// TIA Portal V18 export
// export: Created 2026-06-12T02:00:00Z, ExportSetting WithDefaults
FUNCTION "FC_SCADA_Sim_B3to7" : Void   // FC11, LAD
{ S7_Optimized_Access := 'TRUE' }
VERSION : 0.1
// stored: AutoNumber true, IsIECCheckEnabled false
BEGIN

REGION Network 1: Tạo xung kích hoạt chu kỳ mô phỏng (50ms)
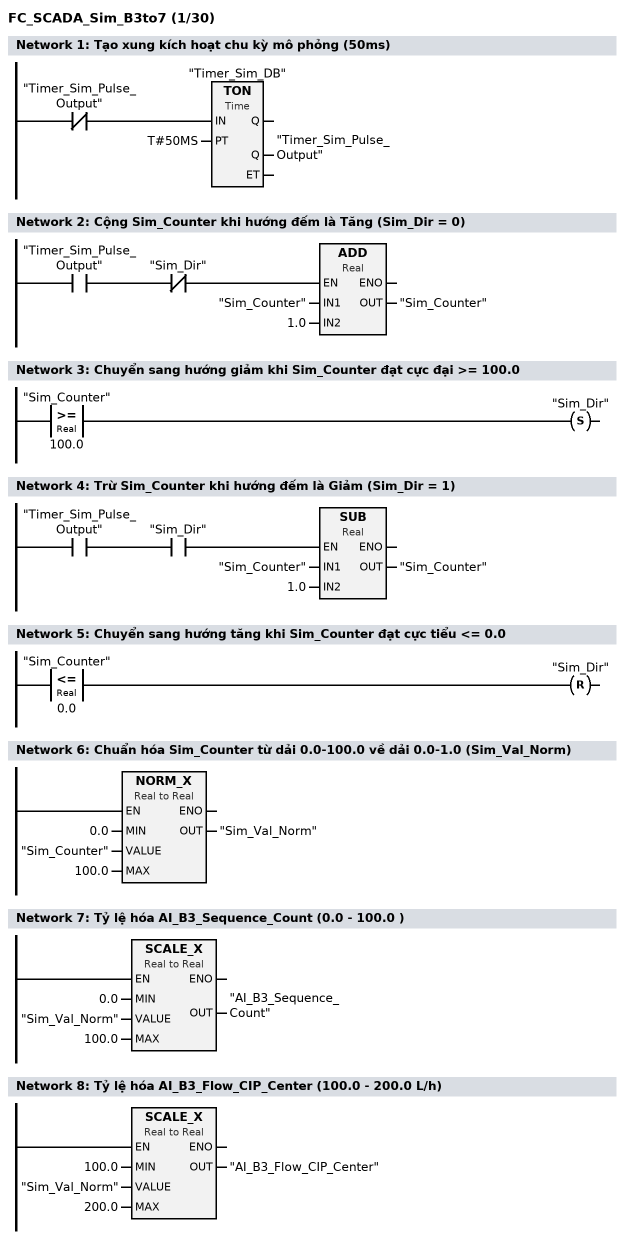
   RUNG wire#powerrail
      I_Contact( "Timer_Sim_Pulse_Output" )
      { S7_Templates := "time_type := Time" } "Timer_Sim_DB".TON(pt := T#50MS, q => "Timer_Sim_Pulse_Output", et =>)
   END_RUNG
   // the same network as SCL:
   "Timer_Sim_DB".TON(IN := NOT "Timer_Sim_Pulse_Output", PT := T#50MS, Q => "Timer_Sim_Pulse_Output");
END_REGION

REGION Network 2: Cộng Sim_Counter khi hướng đếm là Tăng (Sim_Dir = 0)
   RUNG wire#powerrail
      Contact( "Timer_Sim_Pulse_Output" )
      I_Contact( "Sim_Dir" )
      { S7_Templates := "SrcType := Real"; S7_GenerateENO := "TRUE" } Add(in1 := "Sim_Counter", in2 := 1.0, out => "Sim_Counter")
   END_RUNG
   // the same network as SCL:
   IF "Timer_Sim_Pulse_Output" AND NOT "Sim_Dir" THEN "Sim_Counter" := "Sim_Counter" + 1.0; END_IF;
END_REGION

REGION Network 3: Chuyển sang hướng giảm khi Sim_Counter đạt cực đại >= 100.0
   RUNG wire#powerrail
      { S7_Templates := "SrcType := Real" } GE_Contact(in1 := "Sim_Counter", in2 := 100.0)
      S_Coil( "Sim_Dir" )
   END_RUNG
   // the same network as SCL:
   IF "Sim_Counter" >= 100.0 THEN "Sim_Dir" := TRUE; END_IF;
END_REGION

REGION Network 4: Trừ Sim_Counter khi hướng đếm là Giảm (Sim_Dir = 1)
   RUNG wire#powerrail
      Contact( "Timer_Sim_Pulse_Output" )
      Contact( "Sim_Dir" )
      { S7_Templates := "SrcType := Real"; S7_GenerateENO := "TRUE" } Sub(in1 := "Sim_Counter", in2 := 1.0, out => "Sim_Counter")
   END_RUNG
   // the same network as SCL:
   IF "Timer_Sim_Pulse_Output" AND "Sim_Dir" THEN "Sim_Counter" := "Sim_Counter" - 1.0; END_IF;
END_REGION

REGION Network 5: Chuyển sang hướng tăng khi Sim_Counter đạt cực tiểu <= 0.0
   RUNG wire#powerrail
      { S7_Templates := "SrcType := Real" } LE_Contact(in1 := "Sim_Counter", in2 := 0.0)
      R_Coil( "Sim_Dir" )
   END_RUNG
   // the same network as SCL:
   IF "Sim_Counter" <= 0.0 THEN "Sim_Dir" := FALSE; END_IF;
END_REGION

REGION Network 6: Chuẩn hóa Sim_Counter từ dải 0.0-100.0 về dải 0.0-1.0 (Sim_Val_Norm)
   RUNG wire#powerrail
      { S7_Templates := "[SrcType := Real, DestType := Real]" } Normalize(min := 0.0, value := "Sim_Counter", max := 100.0, out => "Sim_Val_Norm")
   END_RUNG
   // the same network as SCL:
   "Sim_Val_Norm" := NORM_X(MIN := 0.0, VALUE := "Sim_Counter", MAX := 100.0);
END_REGION

REGION Network 7: Tỷ lệ hóa AI_B3_Sequence_Count (0.0 - 100.0 )
   RUNG wire#powerrail
      { S7_Templates := "[SrcType := Real, DestType := Real]" } Scale(min := 0.0, value := "Sim_Val_Norm", max := 100.0, out => "AI_B3_Sequence_Count")
   END_RUNG
   // the same network as SCL:
   "AI_B3_Sequence_Count" := SCALE_X(MIN := 0.0, VALUE := "Sim_Val_Norm", MAX := 100.0);
END_REGION

REGION Network 8: Tỷ lệ hóa AI_B3_Flow_CIP_Center (100.0 - 200.0 L/h)
   RUNG wire#powerrail
      { S7_Templates := "[SrcType := Real, DestType := Real]" } Scale(min := 100.0, value := "Sim_Val_Norm", max := 200.0, out => "AI_B3_Flow_CIP_Center")
   END_RUNG
   // the same network as SCL:
   "AI_B3_Flow_CIP_Center" := SCALE_X(MIN := 100.0, VALUE := "Sim_Val_Norm", MAX := 200.0);
END_REGION

REGION Network 9: Tỷ lệ hóa AI_B3_Temp_CIP_Upper (50.0 - 80.0 °C)
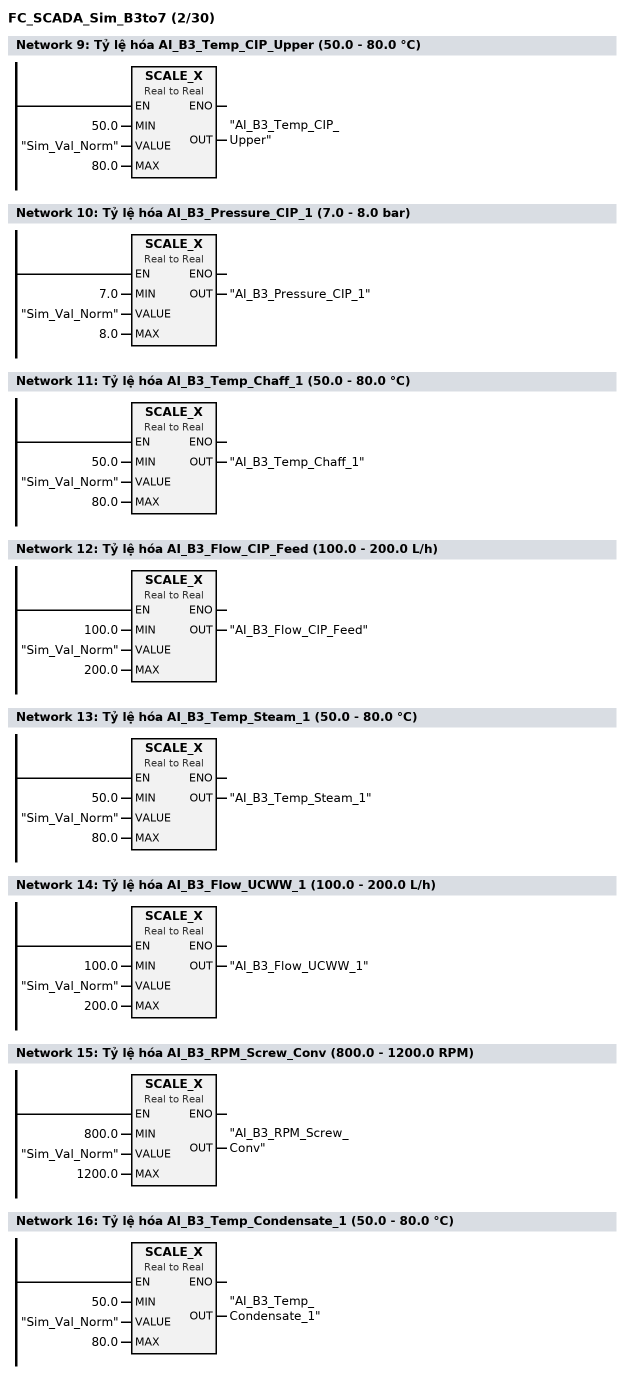
   RUNG wire#powerrail
      { S7_Templates := "[SrcType := Real, DestType := Real]" } Scale(min := 50.0, value := "Sim_Val_Norm", max := 80.0, out => "AI_B3_Temp_CIP_Upper")
   END_RUNG
   // the same network as SCL:
   "AI_B3_Temp_CIP_Upper" := SCALE_X(MIN := 50.0, VALUE := "Sim_Val_Norm", MAX := 80.0);
END_REGION

REGION Network 10: Tỷ lệ hóa AI_B3_Pressure_CIP_1 (7.0 - 8.0 bar)
   RUNG wire#powerrail
      { S7_Templates := "[SrcType := Real, DestType := Real]" } Scale(min := 7.0, value := "Sim_Val_Norm", max := 8.0, out => "AI_B3_Pressure_CIP_1")
   END_RUNG
   // the same network as SCL:
   "AI_B3_Pressure_CIP_1" := SCALE_X(MIN := 7.0, VALUE := "Sim_Val_Norm", MAX := 8.0);
END_REGION

REGION Network 11: Tỷ lệ hóa AI_B3_Temp_Chaff_1 (50.0 - 80.0 °C)
   RUNG wire#powerrail
      { S7_Templates := "[SrcType := Real, DestType := Real]" } Scale(min := 50.0, value := "Sim_Val_Norm", max := 80.0, out => "AI_B3_Temp_Chaff_1")
   END_RUNG
   // the same network as SCL:
   "AI_B3_Temp_Chaff_1" := SCALE_X(MIN := 50.0, VALUE := "Sim_Val_Norm", MAX := 80.0);
END_REGION

REGION Network 12: Tỷ lệ hóa AI_B3_Flow_CIP_Feed (100.0 - 200.0 L/h)
   RUNG wire#powerrail
      { S7_Templates := "[SrcType := Real, DestType := Real]" } Scale(min := 100.0, value := "Sim_Val_Norm", max := 200.0, out => "AI_B3_Flow_CIP_Feed")
   END_RUNG
   // the same network as SCL:
   "AI_B3_Flow_CIP_Feed" := SCALE_X(MIN := 100.0, VALUE := "Sim_Val_Norm", MAX := 200.0);
END_REGION

REGION Network 13: Tỷ lệ hóa AI_B3_Temp_Steam_1 (50.0 - 80.0 °C)
   RUNG wire#powerrail
      { S7_Templates := "[SrcType := Real, DestType := Real]" } Scale(min := 50.0, value := "Sim_Val_Norm", max := 80.0, out => "AI_B3_Temp_Steam_1")
   END_RUNG
   // the same network as SCL:
   "AI_B3_Temp_Steam_1" := SCALE_X(MIN := 50.0, VALUE := "Sim_Val_Norm", MAX := 80.0);
END_REGION

REGION Network 14: Tỷ lệ hóa AI_B3_Flow_UCWW_1 (100.0 - 200.0 L/h)
   RUNG wire#powerrail
      { S7_Templates := "[SrcType := Real, DestType := Real]" } Scale(min := 100.0, value := "Sim_Val_Norm", max := 200.0, out => "AI_B3_Flow_UCWW_1")
   END_RUNG
   // the same network as SCL:
   "AI_B3_Flow_UCWW_1" := SCALE_X(MIN := 100.0, VALUE := "Sim_Val_Norm", MAX := 200.0);
END_REGION

REGION Network 15: Tỷ lệ hóa AI_B3_RPM_Screw_Conv (800.0 - 1200.0 RPM)
   RUNG wire#powerrail
      { S7_Templates := "[SrcType := Real, DestType := Real]" } Scale(min := 800.0, value := "Sim_Val_Norm", max := 1200.0, out => "AI_B3_RPM_Screw_Conv")
   END_RUNG
   // the same network as SCL:
   "AI_B3_RPM_Screw_Conv" := SCALE_X(MIN := 800.0, VALUE := "Sim_Val_Norm", MAX := 1200.0);
END_REGION

REGION Network 16: Tỷ lệ hóa AI_B3_Temp_Condensate_1 (50.0 - 80.0 °C)
   RUNG wire#powerrail
      { S7_Templates := "[SrcType := Real, DestType := Real]" } Scale(min := 50.0, value := "Sim_Val_Norm", max := 80.0, out => "AI_B3_Temp_Condensate_1")
   END_RUNG
   // the same network as SCL:
   "AI_B3_Temp_Condensate_1" := SCALE_X(MIN := 50.0, VALUE := "Sim_Val_Norm", MAX := 80.0);
END_REGION

REGION Network 17: Tỷ lệ hóa AI_B3_Pressure_Screw_1 (7.0 - 8.0 bar)
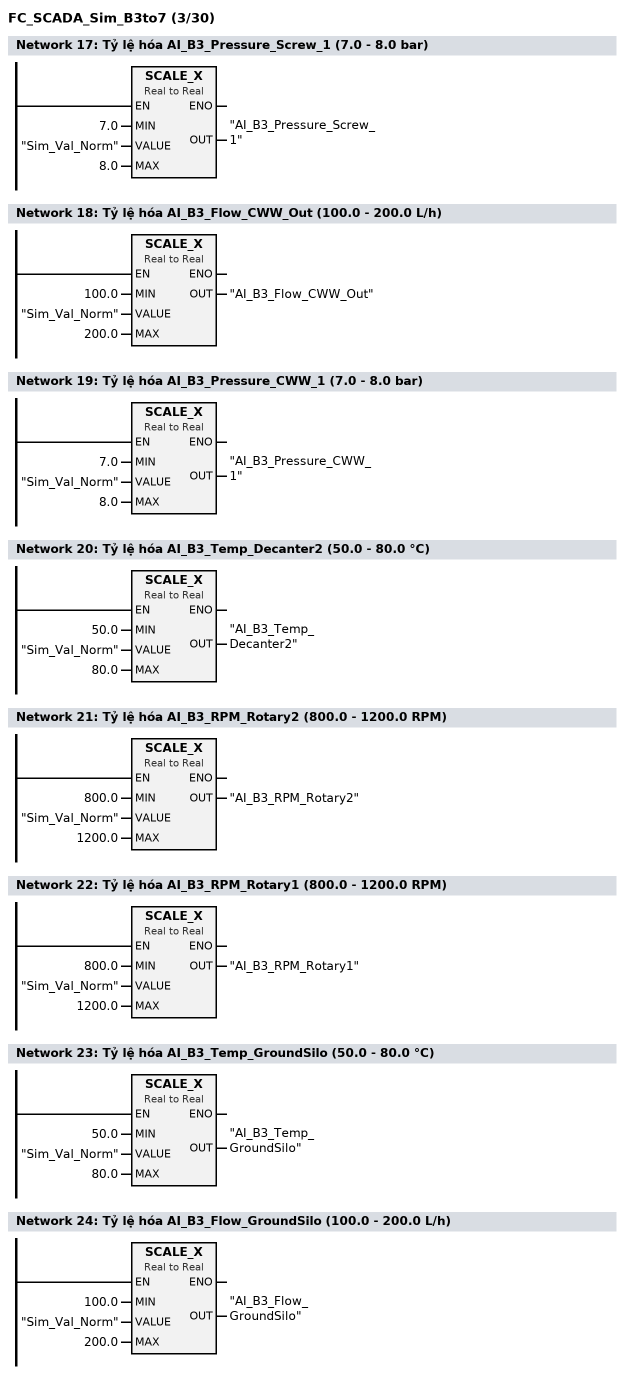
   RUNG wire#powerrail
      { S7_Templates := "[SrcType := Real, DestType := Real]" } Scale(min := 7.0, value := "Sim_Val_Norm", max := 8.0, out => "AI_B3_Pressure_Screw_1")
   END_RUNG
   // the same network as SCL:
   "AI_B3_Pressure_Screw_1" := SCALE_X(MIN := 7.0, VALUE := "Sim_Val_Norm", MAX := 8.0);
END_REGION

REGION Network 18: Tỷ lệ hóa AI_B3_Flow_CWW_Out (100.0 - 200.0 L/h)
   RUNG wire#powerrail
      { S7_Templates := "[SrcType := Real, DestType := Real]" } Scale(min := 100.0, value := "Sim_Val_Norm", max := 200.0, out => "AI_B3_Flow_CWW_Out")
   END_RUNG
   // the same network as SCL:
   "AI_B3_Flow_CWW_Out" := SCALE_X(MIN := 100.0, VALUE := "Sim_Val_Norm", MAX := 200.0);
END_REGION

REGION Network 19: Tỷ lệ hóa AI_B3_Pressure_CWW_1 (7.0 - 8.0 bar)
   RUNG wire#powerrail
      { S7_Templates := "[SrcType := Real, DestType := Real]" } Scale(min := 7.0, value := "Sim_Val_Norm", max := 8.0, out => "AI_B3_Pressure_CWW_1")
   END_RUNG
   // the same network as SCL:
   "AI_B3_Pressure_CWW_1" := SCALE_X(MIN := 7.0, VALUE := "Sim_Val_Norm", MAX := 8.0);
END_REGION

REGION Network 20: Tỷ lệ hóa AI_B3_Temp_Decanter2 (50.0 - 80.0 °C)
   RUNG wire#powerrail
      { S7_Templates := "[SrcType := Real, DestType := Real]" } Scale(min := 50.0, value := "Sim_Val_Norm", max := 80.0, out => "AI_B3_Temp_Decanter2")
   END_RUNG
   // the same network as SCL:
   "AI_B3_Temp_Decanter2" := SCALE_X(MIN := 50.0, VALUE := "Sim_Val_Norm", MAX := 80.0);
END_REGION

REGION Network 21: Tỷ lệ hóa AI_B3_RPM_Rotary2 (800.0 - 1200.0 RPM)
   RUNG wire#powerrail
      { S7_Templates := "[SrcType := Real, DestType := Real]" } Scale(min := 800.0, value := "Sim_Val_Norm", max := 1200.0, out => "AI_B3_RPM_Rotary2")
   END_RUNG
   // the same network as SCL:
   "AI_B3_RPM_Rotary2" := SCALE_X(MIN := 800.0, VALUE := "Sim_Val_Norm", MAX := 1200.0);
END_REGION

REGION Network 22: Tỷ lệ hóa AI_B3_RPM_Rotary1 (800.0 - 1200.0 RPM)
   RUNG wire#powerrail
      { S7_Templates := "[SrcType := Real, DestType := Real]" } Scale(min := 800.0, value := "Sim_Val_Norm", max := 1200.0, out => "AI_B3_RPM_Rotary1")
   END_RUNG
   // the same network as SCL:
   "AI_B3_RPM_Rotary1" := SCALE_X(MIN := 800.0, VALUE := "Sim_Val_Norm", MAX := 1200.0);
END_REGION

REGION Network 23: Tỷ lệ hóa AI_B3_Temp_GroundSilo (50.0 - 80.0 °C)
   RUNG wire#powerrail
      { S7_Templates := "[SrcType := Real, DestType := Real]" } Scale(min := 50.0, value := "Sim_Val_Norm", max := 80.0, out => "AI_B3_Temp_GroundSilo")
   END_RUNG
   // the same network as SCL:
   "AI_B3_Temp_GroundSilo" := SCALE_X(MIN := 50.0, VALUE := "Sim_Val_Norm", MAX := 80.0);
END_REGION

REGION Network 24: Tỷ lệ hóa AI_B3_Flow_GroundSilo (100.0 - 200.0 L/h)
   RUNG wire#powerrail
      { S7_Templates := "[SrcType := Real, DestType := Real]" } Scale(min := 100.0, value := "Sim_Val_Norm", max := 200.0, out => "AI_B3_Flow_GroundSilo")
   END_RUNG
   // the same network as SCL:
   "AI_B3_Flow_GroundSilo" := SCALE_X(MIN := 100.0, VALUE := "Sim_Val_Norm", MAX := 200.0);
END_REGION

REGION Network 25: Tỷ lệ hóa AI_B3_Pressure_Mid_1 (7.0 - 8.0 bar)
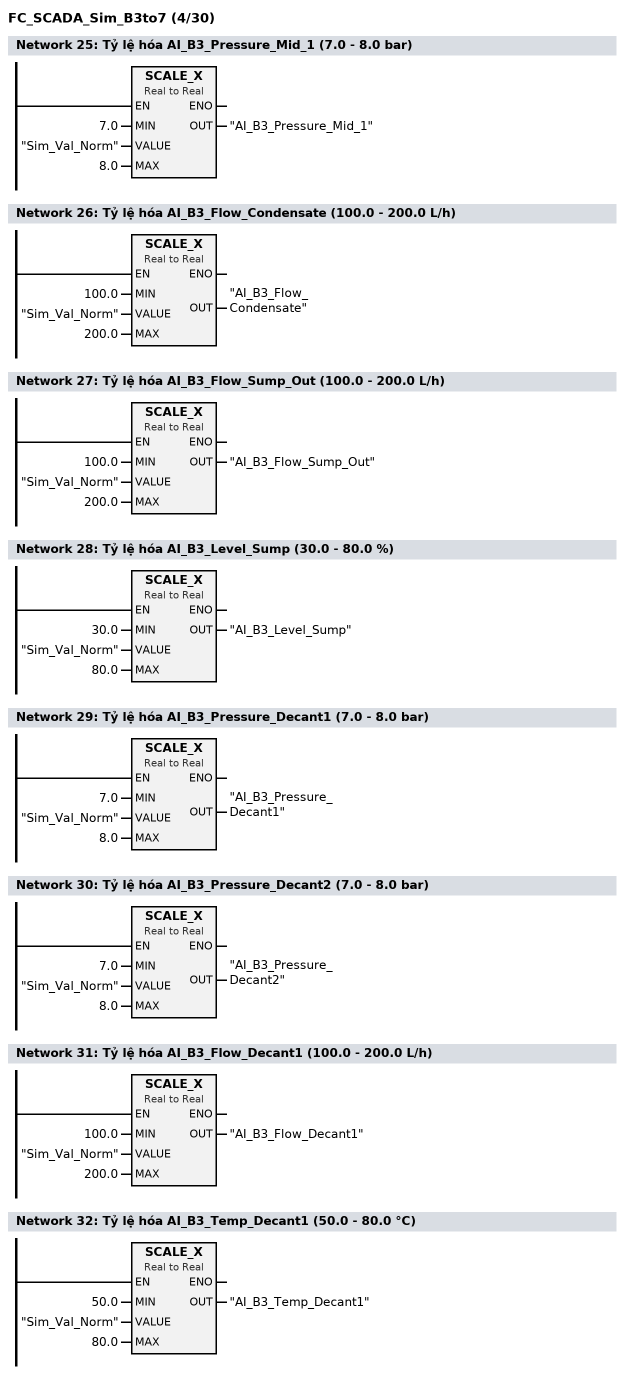
   RUNG wire#powerrail
      { S7_Templates := "[SrcType := Real, DestType := Real]" } Scale(min := 7.0, value := "Sim_Val_Norm", max := 8.0, out => "AI_B3_Pressure_Mid_1")
   END_RUNG
   // the same network as SCL:
   "AI_B3_Pressure_Mid_1" := SCALE_X(MIN := 7.0, VALUE := "Sim_Val_Norm", MAX := 8.0);
END_REGION

REGION Network 26: Tỷ lệ hóa AI_B3_Flow_Condensate (100.0 - 200.0 L/h)
   RUNG wire#powerrail
      { S7_Templates := "[SrcType := Real, DestType := Real]" } Scale(min := 100.0, value := "Sim_Val_Norm", max := 200.0, out => "AI_B3_Flow_Condensate")
   END_RUNG
   // the same network as SCL:
   "AI_B3_Flow_Condensate" := SCALE_X(MIN := 100.0, VALUE := "Sim_Val_Norm", MAX := 200.0);
END_REGION

REGION Network 27: Tỷ lệ hóa AI_B3_Flow_Sump_Out (100.0 - 200.0 L/h)
   RUNG wire#powerrail
      { S7_Templates := "[SrcType := Real, DestType := Real]" } Scale(min := 100.0, value := "Sim_Val_Norm", max := 200.0, out => "AI_B3_Flow_Sump_Out")
   END_RUNG
   // the same network as SCL:
   "AI_B3_Flow_Sump_Out" := SCALE_X(MIN := 100.0, VALUE := "Sim_Val_Norm", MAX := 200.0);
END_REGION

REGION Network 28: Tỷ lệ hóa AI_B3_Level_Sump (30.0 - 80.0 %)
   RUNG wire#powerrail
      { S7_Templates := "[SrcType := Real, DestType := Real]" } Scale(min := 30.0, value := "Sim_Val_Norm", max := 80.0, out => "AI_B3_Level_Sump")
   END_RUNG
   // the same network as SCL:
   "AI_B3_Level_Sump" := SCALE_X(MIN := 30.0, VALUE := "Sim_Val_Norm", MAX := 80.0);
END_REGION

REGION Network 29: Tỷ lệ hóa AI_B3_Pressure_Decant1 (7.0 - 8.0 bar)
   RUNG wire#powerrail
      { S7_Templates := "[SrcType := Real, DestType := Real]" } Scale(min := 7.0, value := "Sim_Val_Norm", max := 8.0, out => "AI_B3_Pressure_Decant1")
   END_RUNG
   // the same network as SCL:
   "AI_B3_Pressure_Decant1" := SCALE_X(MIN := 7.0, VALUE := "Sim_Val_Norm", MAX := 8.0);
END_REGION

REGION Network 30: Tỷ lệ hóa AI_B3_Pressure_Decant2 (7.0 - 8.0 bar)
   RUNG wire#powerrail
      { S7_Templates := "[SrcType := Real, DestType := Real]" } Scale(min := 7.0, value := "Sim_Val_Norm", max := 8.0, out => "AI_B3_Pressure_Decant2")
   END_RUNG
   // the same network as SCL:
   "AI_B3_Pressure_Decant2" := SCALE_X(MIN := 7.0, VALUE := "Sim_Val_Norm", MAX := 8.0);
END_REGION

REGION Network 31: Tỷ lệ hóa AI_B3_Flow_Decant1 (100.0 - 200.0 L/h)
   RUNG wire#powerrail
      { S7_Templates := "[SrcType := Real, DestType := Real]" } Scale(min := 100.0, value := "Sim_Val_Norm", max := 200.0, out => "AI_B3_Flow_Decant1")
   END_RUNG
   // the same network as SCL:
   "AI_B3_Flow_Decant1" := SCALE_X(MIN := 100.0, VALUE := "Sim_Val_Norm", MAX := 200.0);
END_REGION

REGION Network 32: Tỷ lệ hóa AI_B3_Temp_Decant1 (50.0 - 80.0 °C)
   RUNG wire#powerrail
      { S7_Templates := "[SrcType := Real, DestType := Real]" } Scale(min := 50.0, value := "Sim_Val_Norm", max := 80.0, out => "AI_B3_Temp_Decant1")
   END_RUNG
   // the same network as SCL:
   "AI_B3_Temp_Decant1" := SCALE_X(MIN := 50.0, VALUE := "Sim_Val_Norm", MAX := 80.0);
END_REGION

REGION Network 33: Tỷ lệ hóa AI_B3_Temp_FBB_Boiler (50.0 - 80.0 °C)
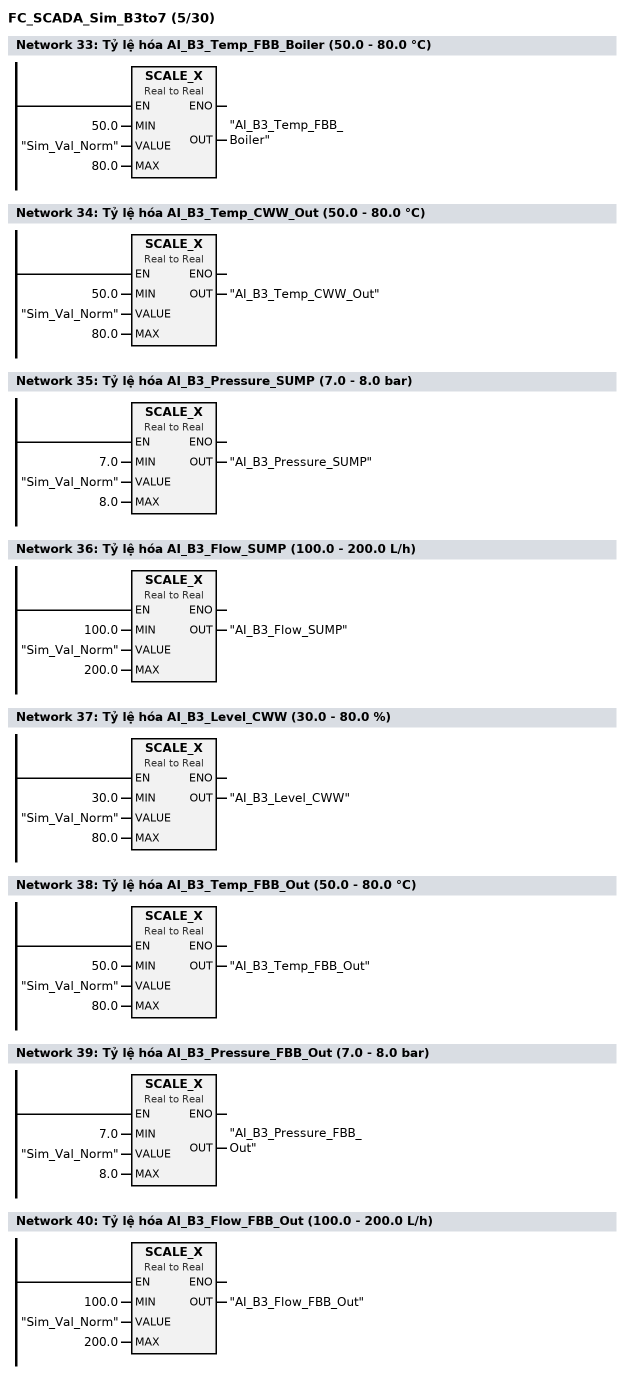
   RUNG wire#powerrail
      { S7_Templates := "[SrcType := Real, DestType := Real]" } Scale(min := 50.0, value := "Sim_Val_Norm", max := 80.0, out => "AI_B3_Temp_FBB_Boiler")
   END_RUNG
   // the same network as SCL:
   "AI_B3_Temp_FBB_Boiler" := SCALE_X(MIN := 50.0, VALUE := "Sim_Val_Norm", MAX := 80.0);
END_REGION

REGION Network 34: Tỷ lệ hóa AI_B3_Temp_CWW_Out (50.0 - 80.0 °C)
   RUNG wire#powerrail
      { S7_Templates := "[SrcType := Real, DestType := Real]" } Scale(min := 50.0, value := "Sim_Val_Norm", max := 80.0, out => "AI_B3_Temp_CWW_Out")
   END_RUNG
   // the same network as SCL:
   "AI_B3_Temp_CWW_Out" := SCALE_X(MIN := 50.0, VALUE := "Sim_Val_Norm", MAX := 80.0);
END_REGION

REGION Network 35: Tỷ lệ hóa AI_B3_Pressure_SUMP (7.0 - 8.0 bar)
   RUNG wire#powerrail
      { S7_Templates := "[SrcType := Real, DestType := Real]" } Scale(min := 7.0, value := "Sim_Val_Norm", max := 8.0, out => "AI_B3_Pressure_SUMP")
   END_RUNG
   // the same network as SCL:
   "AI_B3_Pressure_SUMP" := SCALE_X(MIN := 7.0, VALUE := "Sim_Val_Norm", MAX := 8.0);
END_REGION

REGION Network 36: Tỷ lệ hóa AI_B3_Flow_SUMP (100.0 - 200.0 L/h)
   RUNG wire#powerrail
      { S7_Templates := "[SrcType := Real, DestType := Real]" } Scale(min := 100.0, value := "Sim_Val_Norm", max := 200.0, out => "AI_B3_Flow_SUMP")
   END_RUNG
   // the same network as SCL:
   "AI_B3_Flow_SUMP" := SCALE_X(MIN := 100.0, VALUE := "Sim_Val_Norm", MAX := 200.0);
END_REGION

REGION Network 37: Tỷ lệ hóa AI_B3_Level_CWW (30.0 - 80.0 %)
   RUNG wire#powerrail
      { S7_Templates := "[SrcType := Real, DestType := Real]" } Scale(min := 30.0, value := "Sim_Val_Norm", max := 80.0, out => "AI_B3_Level_CWW")
   END_RUNG
   // the same network as SCL:
   "AI_B3_Level_CWW" := SCALE_X(MIN := 30.0, VALUE := "Sim_Val_Norm", MAX := 80.0);
END_REGION

REGION Network 38: Tỷ lệ hóa AI_B3_Temp_FBB_Out (50.0 - 80.0 °C)
   RUNG wire#powerrail
      { S7_Templates := "[SrcType := Real, DestType := Real]" } Scale(min := 50.0, value := "Sim_Val_Norm", max := 80.0, out => "AI_B3_Temp_FBB_Out")
   END_RUNG
   // the same network as SCL:
   "AI_B3_Temp_FBB_Out" := SCALE_X(MIN := 50.0, VALUE := "Sim_Val_Norm", MAX := 80.0);
END_REGION

REGION Network 39: Tỷ lệ hóa AI_B3_Pressure_FBB_Out (7.0 - 8.0 bar)
   RUNG wire#powerrail
      { S7_Templates := "[SrcType := Real, DestType := Real]" } Scale(min := 7.0, value := "Sim_Val_Norm", max := 8.0, out => "AI_B3_Pressure_FBB_Out")
   END_RUNG
   // the same network as SCL:
   "AI_B3_Pressure_FBB_Out" := SCALE_X(MIN := 7.0, VALUE := "Sim_Val_Norm", MAX := 8.0);
END_REGION

REGION Network 40: Tỷ lệ hóa AI_B3_Flow_FBB_Out (100.0 - 200.0 L/h)
   RUNG wire#powerrail
      { S7_Templates := "[SrcType := Real, DestType := Real]" } Scale(min := 100.0, value := "Sim_Val_Norm", max := 200.0, out => "AI_B3_Flow_FBB_Out")
   END_RUNG
   // the same network as SCL:
   "AI_B3_Flow_FBB_Out" := SCALE_X(MIN := 100.0, VALUE := "Sim_Val_Norm", MAX := 200.0);
END_REGION

REGION Network 41: Tỷ lệ hóa AI_B4_Daq_C (0.0 - 100.0 )
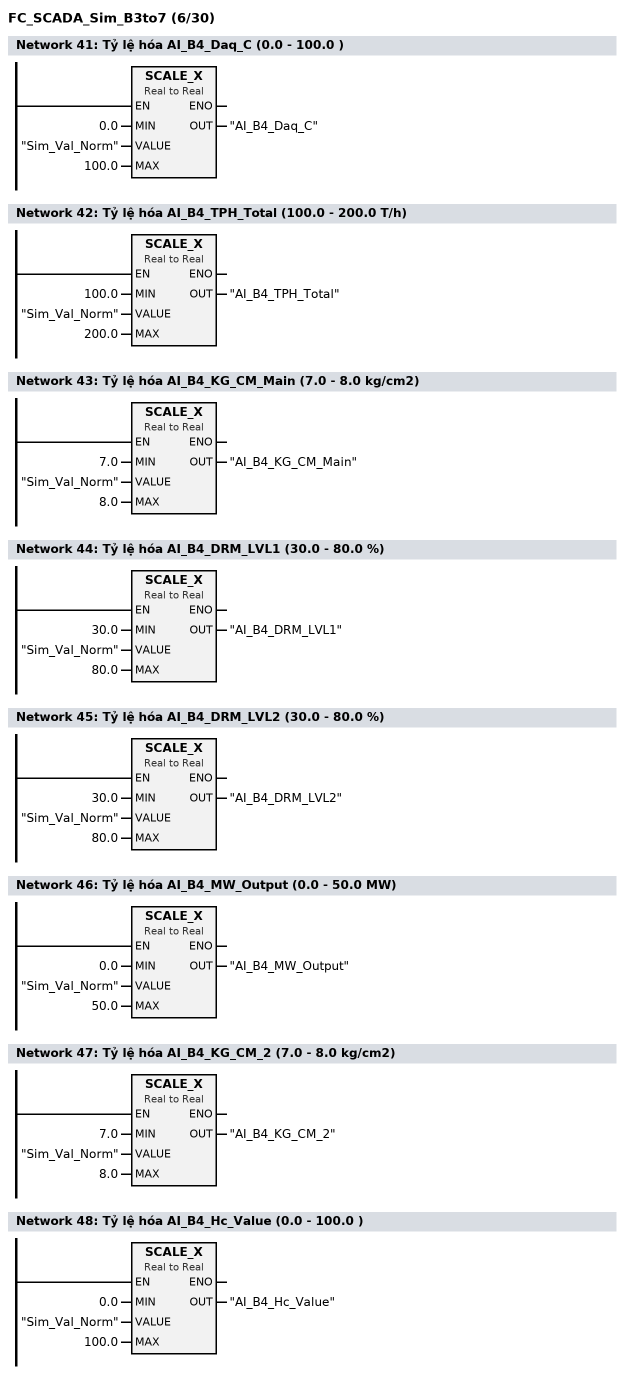
   RUNG wire#powerrail
      { S7_Templates := "[SrcType := Real, DestType := Real]" } Scale(min := 0.0, value := "Sim_Val_Norm", max := 100.0, out => "AI_B4_Daq_C")
   END_RUNG
   // the same network as SCL:
   "AI_B4_Daq_C" := SCALE_X(MIN := 0.0, VALUE := "Sim_Val_Norm", MAX := 100.0);
END_REGION

REGION Network 42: Tỷ lệ hóa AI_B4_TPH_Total (100.0 - 200.0 T/h)
   RUNG wire#powerrail
      { S7_Templates := "[SrcType := Real, DestType := Real]" } Scale(min := 100.0, value := "Sim_Val_Norm", max := 200.0, out => "AI_B4_TPH_Total")
   END_RUNG
   // the same network as SCL:
   "AI_B4_TPH_Total" := SCALE_X(MIN := 100.0, VALUE := "Sim_Val_Norm", MAX := 200.0);
END_REGION

REGION Network 43: Tỷ lệ hóa AI_B4_KG_CM_Main (7.0 - 8.0 kg/cm2)
   RUNG wire#powerrail
      { S7_Templates := "[SrcType := Real, DestType := Real]" } Scale(min := 7.0, value := "Sim_Val_Norm", max := 8.0, out => "AI_B4_KG_CM_Main")
   END_RUNG
   // the same network as SCL:
   "AI_B4_KG_CM_Main" := SCALE_X(MIN := 7.0, VALUE := "Sim_Val_Norm", MAX := 8.0);
END_REGION

REGION Network 44: Tỷ lệ hóa AI_B4_DRM_LVL1 (30.0 - 80.0 %)
   RUNG wire#powerrail
      { S7_Templates := "[SrcType := Real, DestType := Real]" } Scale(min := 30.0, value := "Sim_Val_Norm", max := 80.0, out => "AI_B4_DRM_LVL1")
   END_RUNG
   // the same network as SCL:
   "AI_B4_DRM_LVL1" := SCALE_X(MIN := 30.0, VALUE := "Sim_Val_Norm", MAX := 80.0);
END_REGION

REGION Network 45: Tỷ lệ hóa AI_B4_DRM_LVL2 (30.0 - 80.0 %)
   RUNG wire#powerrail
      { S7_Templates := "[SrcType := Real, DestType := Real]" } Scale(min := 30.0, value := "Sim_Val_Norm", max := 80.0, out => "AI_B4_DRM_LVL2")
   END_RUNG
   // the same network as SCL:
   "AI_B4_DRM_LVL2" := SCALE_X(MIN := 30.0, VALUE := "Sim_Val_Norm", MAX := 80.0);
END_REGION

REGION Network 46: Tỷ lệ hóa AI_B4_MW_Output (0.0 - 50.0 MW)
   RUNG wire#powerrail
      { S7_Templates := "[SrcType := Real, DestType := Real]" } Scale(min := 0.0, value := "Sim_Val_Norm", max := 50.0, out => "AI_B4_MW_Output")
   END_RUNG
   // the same network as SCL:
   "AI_B4_MW_Output" := SCALE_X(MIN := 0.0, VALUE := "Sim_Val_Norm", MAX := 50.0);
END_REGION

REGION Network 47: Tỷ lệ hóa AI_B4_KG_CM_2 (7.0 - 8.0 kg/cm2)
   RUNG wire#powerrail
      { S7_Templates := "[SrcType := Real, DestType := Real]" } Scale(min := 7.0, value := "Sim_Val_Norm", max := 8.0, out => "AI_B4_KG_CM_2")
   END_RUNG
   // the same network as SCL:
   "AI_B4_KG_CM_2" := SCALE_X(MIN := 7.0, VALUE := "Sim_Val_Norm", MAX := 8.0);
END_REGION

REGION Network 48: Tỷ lệ hóa AI_B4_Hc_Value (0.0 - 100.0 )
   RUNG wire#powerrail
      { S7_Templates := "[SrcType := Real, DestType := Real]" } Scale(min := 0.0, value := "Sim_Val_Norm", max := 100.0, out => "AI_B4_Hc_Value")
   END_RUNG
   // the same network as SCL:
   "AI_B4_Hc_Value" := SCALE_X(MIN := 0.0, VALUE := "Sim_Val_Norm", MAX := 100.0);
END_REGION

REGION Network 49: Tỷ lệ hóa AI_B4_Temp_AirHeater_In1 (50.0 - 80.0 °C)
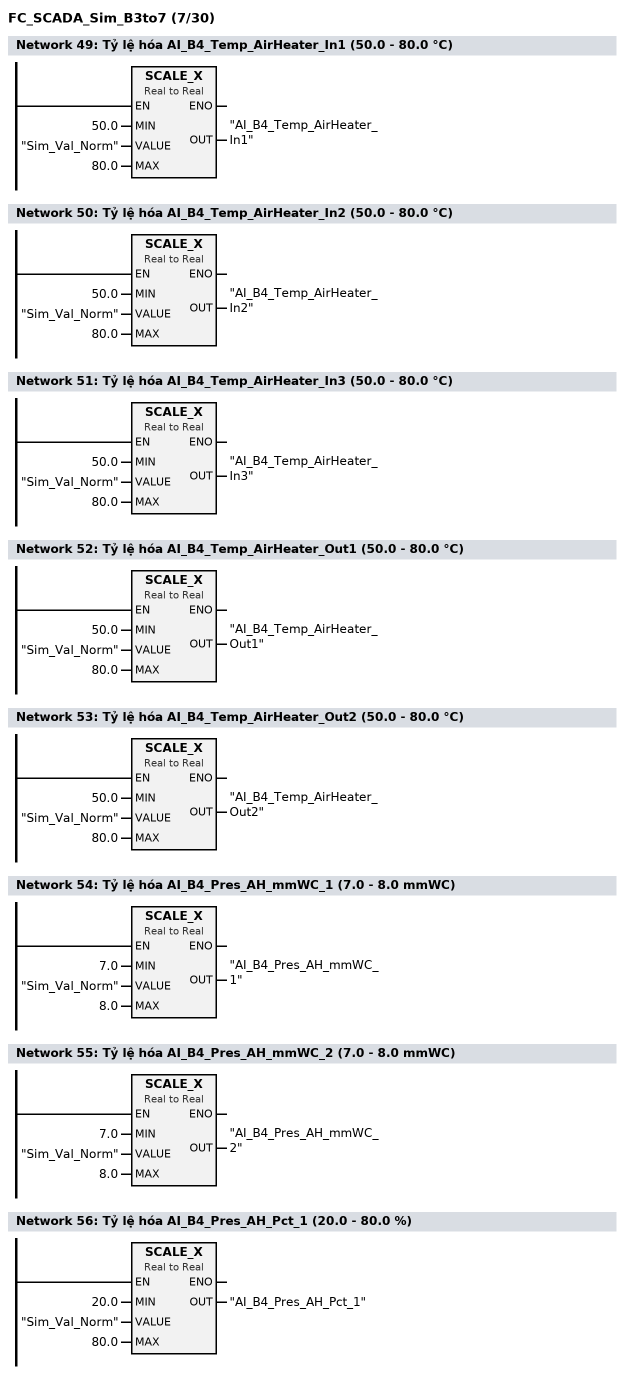
   RUNG wire#powerrail
      { S7_Templates := "[SrcType := Real, DestType := Real]" } Scale(min := 50.0, value := "Sim_Val_Norm", max := 80.0, out => "AI_B4_Temp_AirHeater_In1")
   END_RUNG
   // the same network as SCL:
   "AI_B4_Temp_AirHeater_In1" := SCALE_X(MIN := 50.0, VALUE := "Sim_Val_Norm", MAX := 80.0);
END_REGION

REGION Network 50: Tỷ lệ hóa AI_B4_Temp_AirHeater_In2 (50.0 - 80.0 °C)
   RUNG wire#powerrail
      { S7_Templates := "[SrcType := Real, DestType := Real]" } Scale(min := 50.0, value := "Sim_Val_Norm", max := 80.0, out => "AI_B4_Temp_AirHeater_In2")
   END_RUNG
   // the same network as SCL:
   "AI_B4_Temp_AirHeater_In2" := SCALE_X(MIN := 50.0, VALUE := "Sim_Val_Norm", MAX := 80.0);
END_REGION

REGION Network 51: Tỷ lệ hóa AI_B4_Temp_AirHeater_In3 (50.0 - 80.0 °C)
   RUNG wire#powerrail
      { S7_Templates := "[SrcType := Real, DestType := Real]" } Scale(min := 50.0, value := "Sim_Val_Norm", max := 80.0, out => "AI_B4_Temp_AirHeater_In3")
   END_RUNG
   // the same network as SCL:
   "AI_B4_Temp_AirHeater_In3" := SCALE_X(MIN := 50.0, VALUE := "Sim_Val_Norm", MAX := 80.0);
END_REGION

REGION Network 52: Tỷ lệ hóa AI_B4_Temp_AirHeater_Out1 (50.0 - 80.0 °C)
   RUNG wire#powerrail
      { S7_Templates := "[SrcType := Real, DestType := Real]" } Scale(min := 50.0, value := "Sim_Val_Norm", max := 80.0, out => "AI_B4_Temp_AirHeater_Out1")
   END_RUNG
   // the same network as SCL:
   "AI_B4_Temp_AirHeater_Out1" := SCALE_X(MIN := 50.0, VALUE := "Sim_Val_Norm", MAX := 80.0);
END_REGION

REGION Network 53: Tỷ lệ hóa AI_B4_Temp_AirHeater_Out2 (50.0 - 80.0 °C)
   RUNG wire#powerrail
      { S7_Templates := "[SrcType := Real, DestType := Real]" } Scale(min := 50.0, value := "Sim_Val_Norm", max := 80.0, out => "AI_B4_Temp_AirHeater_Out2")
   END_RUNG
   // the same network as SCL:
   "AI_B4_Temp_AirHeater_Out2" := SCALE_X(MIN := 50.0, VALUE := "Sim_Val_Norm", MAX := 80.0);
END_REGION

REGION Network 54: Tỷ lệ hóa AI_B4_Pres_AH_mmWC_1 (7.0 - 8.0 mmWC)
   RUNG wire#powerrail
      { S7_Templates := "[SrcType := Real, DestType := Real]" } Scale(min := 7.0, value := "Sim_Val_Norm", max := 8.0, out => "AI_B4_Pres_AH_mmWC_1")
   END_RUNG
   // the same network as SCL:
   "AI_B4_Pres_AH_mmWC_1" := SCALE_X(MIN := 7.0, VALUE := "Sim_Val_Norm", MAX := 8.0);
END_REGION

REGION Network 55: Tỷ lệ hóa AI_B4_Pres_AH_mmWC_2 (7.0 - 8.0 mmWC)
   RUNG wire#powerrail
      { S7_Templates := "[SrcType := Real, DestType := Real]" } Scale(min := 7.0, value := "Sim_Val_Norm", max := 8.0, out => "AI_B4_Pres_AH_mmWC_2")
   END_RUNG
   // the same network as SCL:
   "AI_B4_Pres_AH_mmWC_2" := SCALE_X(MIN := 7.0, VALUE := "Sim_Val_Norm", MAX := 8.0);
END_REGION

REGION Network 56: Tỷ lệ hóa AI_B4_Pres_AH_Pct_1 (20.0 - 80.0 %)
   RUNG wire#powerrail
      { S7_Templates := "[SrcType := Real, DestType := Real]" } Scale(min := 20.0, value := "Sim_Val_Norm", max := 80.0, out => "AI_B4_Pres_AH_Pct_1")
   END_RUNG
   // the same network as SCL:
   "AI_B4_Pres_AH_Pct_1" := SCALE_X(MIN := 20.0, VALUE := "Sim_Val_Norm", MAX := 80.0);
END_REGION

REGION Network 57: Tỷ lệ hóa AI_B4_Temp_AH_Out3 (50.0 - 80.0 °C)
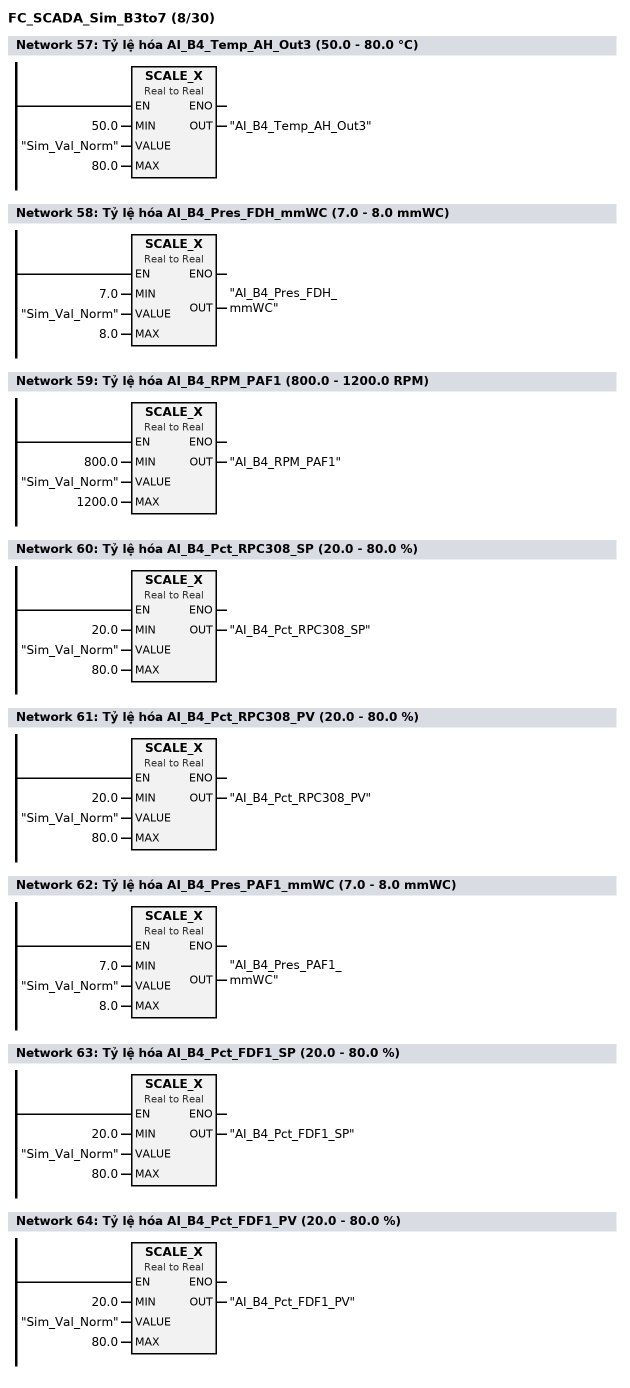
   RUNG wire#powerrail
      { S7_Templates := "[SrcType := Real, DestType := Real]" } Scale(min := 50.0, value := "Sim_Val_Norm", max := 80.0, out => "AI_B4_Temp_AH_Out3")
   END_RUNG
   // the same network as SCL:
   "AI_B4_Temp_AH_Out3" := SCALE_X(MIN := 50.0, VALUE := "Sim_Val_Norm", MAX := 80.0);
END_REGION

REGION Network 58: Tỷ lệ hóa AI_B4_Pres_FDH_mmWC (7.0 - 8.0 mmWC)
   RUNG wire#powerrail
      { S7_Templates := "[SrcType := Real, DestType := Real]" } Scale(min := 7.0, value := "Sim_Val_Norm", max := 8.0, out => "AI_B4_Pres_FDH_mmWC")
   END_RUNG
   // the same network as SCL:
   "AI_B4_Pres_FDH_mmWC" := SCALE_X(MIN := 7.0, VALUE := "Sim_Val_Norm", MAX := 8.0);
END_REGION

REGION Network 59: Tỷ lệ hóa AI_B4_RPM_PAF1 (800.0 - 1200.0 RPM)
   RUNG wire#powerrail
      { S7_Templates := "[SrcType := Real, DestType := Real]" } Scale(min := 800.0, value := "Sim_Val_Norm", max := 1200.0, out => "AI_B4_RPM_PAF1")
   END_RUNG
   // the same network as SCL:
   "AI_B4_RPM_PAF1" := SCALE_X(MIN := 800.0, VALUE := "Sim_Val_Norm", MAX := 1200.0);
END_REGION

REGION Network 60: Tỷ lệ hóa AI_B4_Pct_RPC308_SP (20.0 - 80.0 %)
   RUNG wire#powerrail
      { S7_Templates := "[SrcType := Real, DestType := Real]" } Scale(min := 20.0, value := "Sim_Val_Norm", max := 80.0, out => "AI_B4_Pct_RPC308_SP")
   END_RUNG
   // the same network as SCL:
   "AI_B4_Pct_RPC308_SP" := SCALE_X(MIN := 20.0, VALUE := "Sim_Val_Norm", MAX := 80.0);
END_REGION

REGION Network 61: Tỷ lệ hóa AI_B4_Pct_RPC308_PV (20.0 - 80.0 %)
   RUNG wire#powerrail
      { S7_Templates := "[SrcType := Real, DestType := Real]" } Scale(min := 20.0, value := "Sim_Val_Norm", max := 80.0, out => "AI_B4_Pct_RPC308_PV")
   END_RUNG
   // the same network as SCL:
   "AI_B4_Pct_RPC308_PV" := SCALE_X(MIN := 20.0, VALUE := "Sim_Val_Norm", MAX := 80.0);
END_REGION

REGION Network 62: Tỷ lệ hóa AI_B4_Pres_PAF1_mmWC (7.0 - 8.0 mmWC)
   RUNG wire#powerrail
      { S7_Templates := "[SrcType := Real, DestType := Real]" } Scale(min := 7.0, value := "Sim_Val_Norm", max := 8.0, out => "AI_B4_Pres_PAF1_mmWC")
   END_RUNG
   // the same network as SCL:
   "AI_B4_Pres_PAF1_mmWC" := SCALE_X(MIN := 7.0, VALUE := "Sim_Val_Norm", MAX := 8.0);
END_REGION

REGION Network 63: Tỷ lệ hóa AI_B4_Pct_FDF1_SP (20.0 - 80.0 %)
   RUNG wire#powerrail
      { S7_Templates := "[SrcType := Real, DestType := Real]" } Scale(min := 20.0, value := "Sim_Val_Norm", max := 80.0, out => "AI_B4_Pct_FDF1_SP")
   END_RUNG
   // the same network as SCL:
   "AI_B4_Pct_FDF1_SP" := SCALE_X(MIN := 20.0, VALUE := "Sim_Val_Norm", MAX := 80.0);
END_REGION

REGION Network 64: Tỷ lệ hóa AI_B4_Pct_FDF1_PV (20.0 - 80.0 %)
   RUNG wire#powerrail
      { S7_Templates := "[SrcType := Real, DestType := Real]" } Scale(min := 20.0, value := "Sim_Val_Norm", max := 80.0, out => "AI_B4_Pct_FDF1_PV")
   END_RUNG
   // the same network as SCL:
   "AI_B4_Pct_FDF1_PV" := SCALE_X(MIN := 20.0, VALUE := "Sim_Val_Norm", MAX := 80.0);
END_REGION

REGION Network 65: Tỷ lệ hóa AI_B4_Pct_FDF1_OUT (20.0 - 80.0 %)
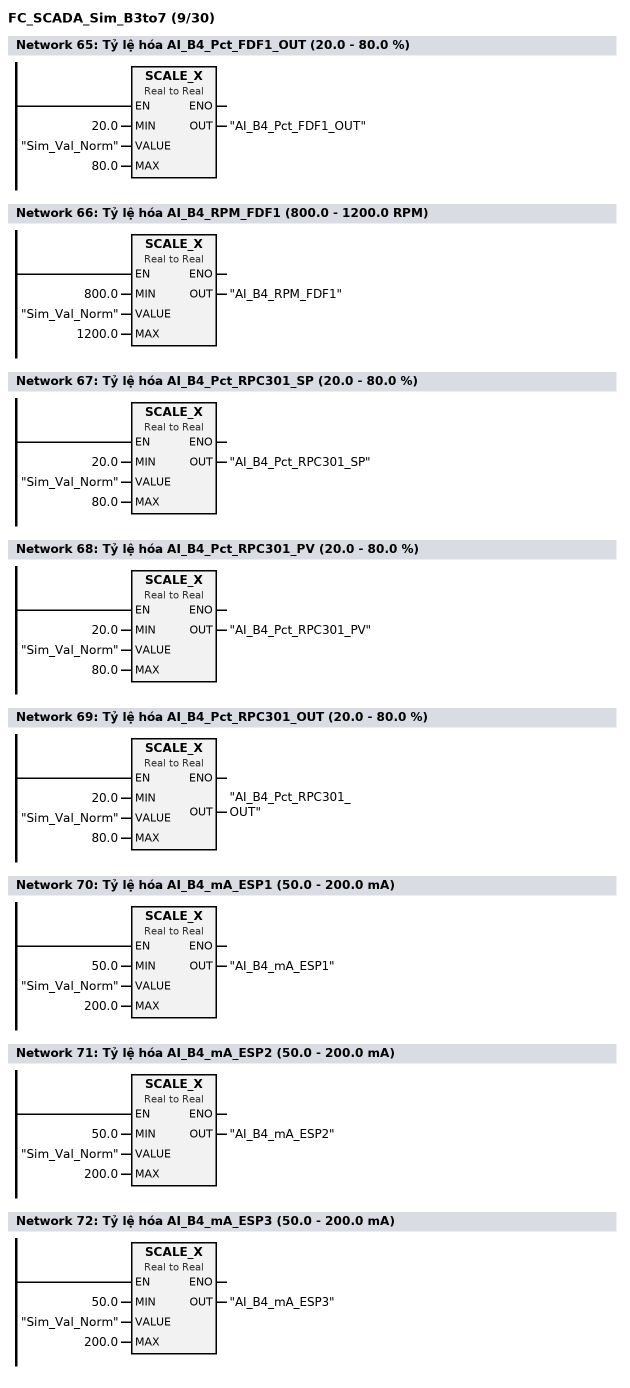
   RUNG wire#powerrail
      { S7_Templates := "[SrcType := Real, DestType := Real]" } Scale(min := 20.0, value := "Sim_Val_Norm", max := 80.0, out => "AI_B4_Pct_FDF1_OUT")
   END_RUNG
   // the same network as SCL:
   "AI_B4_Pct_FDF1_OUT" := SCALE_X(MIN := 20.0, VALUE := "Sim_Val_Norm", MAX := 80.0);
END_REGION

REGION Network 66: Tỷ lệ hóa AI_B4_RPM_FDF1 (800.0 - 1200.0 RPM)
   RUNG wire#powerrail
      { S7_Templates := "[SrcType := Real, DestType := Real]" } Scale(min := 800.0, value := "Sim_Val_Norm", max := 1200.0, out => "AI_B4_RPM_FDF1")
   END_RUNG
   // the same network as SCL:
   "AI_B4_RPM_FDF1" := SCALE_X(MIN := 800.0, VALUE := "Sim_Val_Norm", MAX := 1200.0);
END_REGION

REGION Network 67: Tỷ lệ hóa AI_B4_Pct_RPC301_SP (20.0 - 80.0 %)
   RUNG wire#powerrail
      { S7_Templates := "[SrcType := Real, DestType := Real]" } Scale(min := 20.0, value := "Sim_Val_Norm", max := 80.0, out => "AI_B4_Pct_RPC301_SP")
   END_RUNG
   // the same network as SCL:
   "AI_B4_Pct_RPC301_SP" := SCALE_X(MIN := 20.0, VALUE := "Sim_Val_Norm", MAX := 80.0);
END_REGION

REGION Network 68: Tỷ lệ hóa AI_B4_Pct_RPC301_PV (20.0 - 80.0 %)
   RUNG wire#powerrail
      { S7_Templates := "[SrcType := Real, DestType := Real]" } Scale(min := 20.0, value := "Sim_Val_Norm", max := 80.0, out => "AI_B4_Pct_RPC301_PV")
   END_RUNG
   // the same network as SCL:
   "AI_B4_Pct_RPC301_PV" := SCALE_X(MIN := 20.0, VALUE := "Sim_Val_Norm", MAX := 80.0);
END_REGION

REGION Network 69: Tỷ lệ hóa AI_B4_Pct_RPC301_OUT (20.0 - 80.0 %)
   RUNG wire#powerrail
      { S7_Templates := "[SrcType := Real, DestType := Real]" } Scale(min := 20.0, value := "Sim_Val_Norm", max := 80.0, out => "AI_B4_Pct_RPC301_OUT")
   END_RUNG
   // the same network as SCL:
   "AI_B4_Pct_RPC301_OUT" := SCALE_X(MIN := 20.0, VALUE := "Sim_Val_Norm", MAX := 80.0);
END_REGION

REGION Network 70: Tỷ lệ hóa AI_B4_mA_ESP1 (50.0 - 200.0 mA)
   RUNG wire#powerrail
      { S7_Templates := "[SrcType := Real, DestType := Real]" } Scale(min := 50.0, value := "Sim_Val_Norm", max := 200.0, out => "AI_B4_mA_ESP1")
   END_RUNG
   // the same network as SCL:
   "AI_B4_mA_ESP1" := SCALE_X(MIN := 50.0, VALUE := "Sim_Val_Norm", MAX := 200.0);
END_REGION

REGION Network 71: Tỷ lệ hóa AI_B4_mA_ESP2 (50.0 - 200.0 mA)
   RUNG wire#powerrail
      { S7_Templates := "[SrcType := Real, DestType := Real]" } Scale(min := 50.0, value := "Sim_Val_Norm", max := 200.0, out => "AI_B4_mA_ESP2")
   END_RUNG
   // the same network as SCL:
   "AI_B4_mA_ESP2" := SCALE_X(MIN := 50.0, VALUE := "Sim_Val_Norm", MAX := 200.0);
END_REGION

REGION Network 72: Tỷ lệ hóa AI_B4_mA_ESP3 (50.0 - 200.0 mA)
   RUNG wire#powerrail
      { S7_Templates := "[SrcType := Real, DestType := Real]" } Scale(min := 50.0, value := "Sim_Val_Norm", max := 200.0, out => "AI_B4_mA_ESP3")
   END_RUNG
   // the same network as SCL:
   "AI_B4_mA_ESP3" := SCALE_X(MIN := 50.0, VALUE := "Sim_Val_Norm", MAX := 200.0);
END_REGION

REGION Network 73: Tỷ lệ hóa AI_B4_mA_ESP4 (50.0 - 200.0 mA)
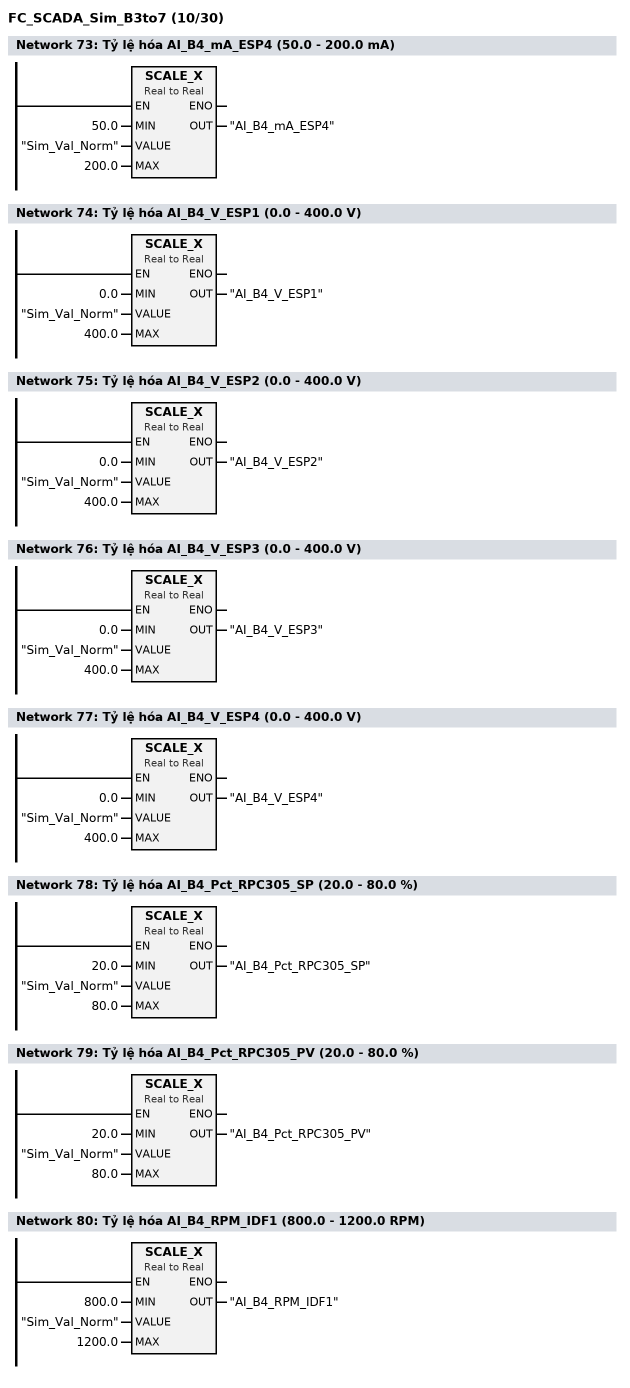
   RUNG wire#powerrail
      { S7_Templates := "[SrcType := Real, DestType := Real]" } Scale(min := 50.0, value := "Sim_Val_Norm", max := 200.0, out => "AI_B4_mA_ESP4")
   END_RUNG
   // the same network as SCL:
   "AI_B4_mA_ESP4" := SCALE_X(MIN := 50.0, VALUE := "Sim_Val_Norm", MAX := 200.0);
END_REGION

REGION Network 74: Tỷ lệ hóa AI_B4_V_ESP1 (0.0 - 400.0 V)
   RUNG wire#powerrail
      { S7_Templates := "[SrcType := Real, DestType := Real]" } Scale(min := 0.0, value := "Sim_Val_Norm", max := 400.0, out => "AI_B4_V_ESP1")
   END_RUNG
   // the same network as SCL:
   "AI_B4_V_ESP1" := SCALE_X(MIN := 0.0, VALUE := "Sim_Val_Norm", MAX := 400.0);
END_REGION

REGION Network 75: Tỷ lệ hóa AI_B4_V_ESP2 (0.0 - 400.0 V)
   RUNG wire#powerrail
      { S7_Templates := "[SrcType := Real, DestType := Real]" } Scale(min := 0.0, value := "Sim_Val_Norm", max := 400.0, out => "AI_B4_V_ESP2")
   END_RUNG
   // the same network as SCL:
   "AI_B4_V_ESP2" := SCALE_X(MIN := 0.0, VALUE := "Sim_Val_Norm", MAX := 400.0);
END_REGION

REGION Network 76: Tỷ lệ hóa AI_B4_V_ESP3 (0.0 - 400.0 V)
   RUNG wire#powerrail
      { S7_Templates := "[SrcType := Real, DestType := Real]" } Scale(min := 0.0, value := "Sim_Val_Norm", max := 400.0, out => "AI_B4_V_ESP3")
   END_RUNG
   // the same network as SCL:
   "AI_B4_V_ESP3" := SCALE_X(MIN := 0.0, VALUE := "Sim_Val_Norm", MAX := 400.0);
END_REGION

REGION Network 77: Tỷ lệ hóa AI_B4_V_ESP4 (0.0 - 400.0 V)
   RUNG wire#powerrail
      { S7_Templates := "[SrcType := Real, DestType := Real]" } Scale(min := 0.0, value := "Sim_Val_Norm", max := 400.0, out => "AI_B4_V_ESP4")
   END_RUNG
   // the same network as SCL:
   "AI_B4_V_ESP4" := SCALE_X(MIN := 0.0, VALUE := "Sim_Val_Norm", MAX := 400.0);
END_REGION

REGION Network 78: Tỷ lệ hóa AI_B4_Pct_RPC305_SP (20.0 - 80.0 %)
   RUNG wire#powerrail
      { S7_Templates := "[SrcType := Real, DestType := Real]" } Scale(min := 20.0, value := "Sim_Val_Norm", max := 80.0, out => "AI_B4_Pct_RPC305_SP")
   END_RUNG
   // the same network as SCL:
   "AI_B4_Pct_RPC305_SP" := SCALE_X(MIN := 20.0, VALUE := "Sim_Val_Norm", MAX := 80.0);
END_REGION

REGION Network 79: Tỷ lệ hóa AI_B4_Pct_RPC305_PV (20.0 - 80.0 %)
   RUNG wire#powerrail
      { S7_Templates := "[SrcType := Real, DestType := Real]" } Scale(min := 20.0, value := "Sim_Val_Norm", max := 80.0, out => "AI_B4_Pct_RPC305_PV")
   END_RUNG
   // the same network as SCL:
   "AI_B4_Pct_RPC305_PV" := SCALE_X(MIN := 20.0, VALUE := "Sim_Val_Norm", MAX := 80.0);
END_REGION

REGION Network 80: Tỷ lệ hóa AI_B4_RPM_IDF1 (800.0 - 1200.0 RPM)
   RUNG wire#powerrail
      { S7_Templates := "[SrcType := Real, DestType := Real]" } Scale(min := 800.0, value := "Sim_Val_Norm", max := 1200.0, out => "AI_B4_RPM_IDF1")
   END_RUNG
   // the same network as SCL:
   "AI_B4_RPM_IDF1" := SCALE_X(MIN := 800.0, VALUE := "Sim_Val_Norm", MAX := 1200.0);
END_REGION

REGION Network 81: Tỷ lệ hóa AI_B4_Pct_RPC305_VFD (20.0 - 80.0 %)
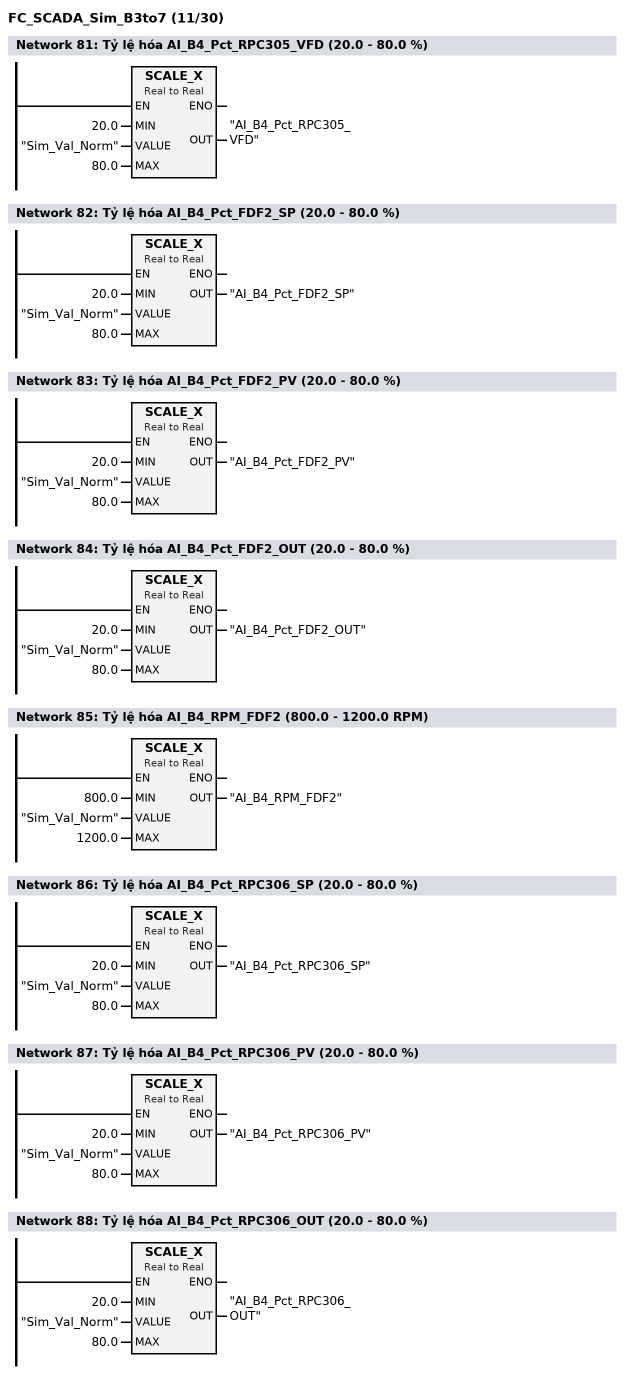
   RUNG wire#powerrail
      { S7_Templates := "[SrcType := Real, DestType := Real]" } Scale(min := 20.0, value := "Sim_Val_Norm", max := 80.0, out => "AI_B4_Pct_RPC305_VFD")
   END_RUNG
   // the same network as SCL:
   "AI_B4_Pct_RPC305_VFD" := SCALE_X(MIN := 20.0, VALUE := "Sim_Val_Norm", MAX := 80.0);
END_REGION

REGION Network 82: Tỷ lệ hóa AI_B4_Pct_FDF2_SP (20.0 - 80.0 %)
   RUNG wire#powerrail
      { S7_Templates := "[SrcType := Real, DestType := Real]" } Scale(min := 20.0, value := "Sim_Val_Norm", max := 80.0, out => "AI_B4_Pct_FDF2_SP")
   END_RUNG
   // the same network as SCL:
   "AI_B4_Pct_FDF2_SP" := SCALE_X(MIN := 20.0, VALUE := "Sim_Val_Norm", MAX := 80.0);
END_REGION

REGION Network 83: Tỷ lệ hóa AI_B4_Pct_FDF2_PV (20.0 - 80.0 %)
   RUNG wire#powerrail
      { S7_Templates := "[SrcType := Real, DestType := Real]" } Scale(min := 20.0, value := "Sim_Val_Norm", max := 80.0, out => "AI_B4_Pct_FDF2_PV")
   END_RUNG
   // the same network as SCL:
   "AI_B4_Pct_FDF2_PV" := SCALE_X(MIN := 20.0, VALUE := "Sim_Val_Norm", MAX := 80.0);
END_REGION

REGION Network 84: Tỷ lệ hóa AI_B4_Pct_FDF2_OUT (20.0 - 80.0 %)
   RUNG wire#powerrail
      { S7_Templates := "[SrcType := Real, DestType := Real]" } Scale(min := 20.0, value := "Sim_Val_Norm", max := 80.0, out => "AI_B4_Pct_FDF2_OUT")
   END_RUNG
   // the same network as SCL:
   "AI_B4_Pct_FDF2_OUT" := SCALE_X(MIN := 20.0, VALUE := "Sim_Val_Norm", MAX := 80.0);
END_REGION

REGION Network 85: Tỷ lệ hóa AI_B4_RPM_FDF2 (800.0 - 1200.0 RPM)
   RUNG wire#powerrail
      { S7_Templates := "[SrcType := Real, DestType := Real]" } Scale(min := 800.0, value := "Sim_Val_Norm", max := 1200.0, out => "AI_B4_RPM_FDF2")
   END_RUNG
   // the same network as SCL:
   "AI_B4_RPM_FDF2" := SCALE_X(MIN := 800.0, VALUE := "Sim_Val_Norm", MAX := 1200.0);
END_REGION

REGION Network 86: Tỷ lệ hóa AI_B4_Pct_RPC306_SP (20.0 - 80.0 %)
   RUNG wire#powerrail
      { S7_Templates := "[SrcType := Real, DestType := Real]" } Scale(min := 20.0, value := "Sim_Val_Norm", max := 80.0, out => "AI_B4_Pct_RPC306_SP")
   END_RUNG
   // the same network as SCL:
   "AI_B4_Pct_RPC306_SP" := SCALE_X(MIN := 20.0, VALUE := "Sim_Val_Norm", MAX := 80.0);
END_REGION

REGION Network 87: Tỷ lệ hóa AI_B4_Pct_RPC306_PV (20.0 - 80.0 %)
   RUNG wire#powerrail
      { S7_Templates := "[SrcType := Real, DestType := Real]" } Scale(min := 20.0, value := "Sim_Val_Norm", max := 80.0, out => "AI_B4_Pct_RPC306_PV")
   END_RUNG
   // the same network as SCL:
   "AI_B4_Pct_RPC306_PV" := SCALE_X(MIN := 20.0, VALUE := "Sim_Val_Norm", MAX := 80.0);
END_REGION

REGION Network 88: Tỷ lệ hóa AI_B4_Pct_RPC306_OUT (20.0 - 80.0 %)
   RUNG wire#powerrail
      { S7_Templates := "[SrcType := Real, DestType := Real]" } Scale(min := 20.0, value := "Sim_Val_Norm", max := 80.0, out => "AI_B4_Pct_RPC306_OUT")
   END_RUNG
   // the same network as SCL:
   "AI_B4_Pct_RPC306_OUT" := SCALE_X(MIN := 20.0, VALUE := "Sim_Val_Norm", MAX := 80.0);
END_REGION

REGION Network 89: Tỷ lệ hóa AI_B4_RPM_IDF2 (800.0 - 1200.0 RPM)
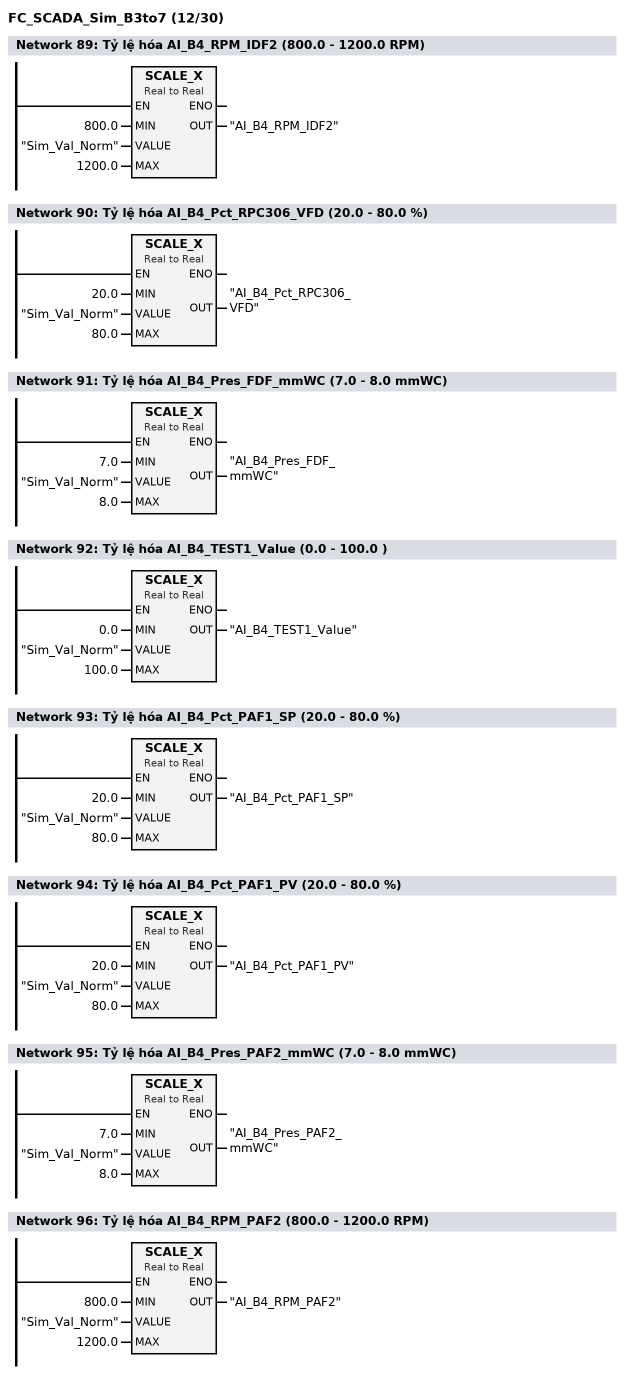
   RUNG wire#powerrail
      { S7_Templates := "[SrcType := Real, DestType := Real]" } Scale(min := 800.0, value := "Sim_Val_Norm", max := 1200.0, out => "AI_B4_RPM_IDF2")
   END_RUNG
   // the same network as SCL:
   "AI_B4_RPM_IDF2" := SCALE_X(MIN := 800.0, VALUE := "Sim_Val_Norm", MAX := 1200.0);
END_REGION

REGION Network 90: Tỷ lệ hóa AI_B4_Pct_RPC306_VFD (20.0 - 80.0 %)
   RUNG wire#powerrail
      { S7_Templates := "[SrcType := Real, DestType := Real]" } Scale(min := 20.0, value := "Sim_Val_Norm", max := 80.0, out => "AI_B4_Pct_RPC306_VFD")
   END_RUNG
   // the same network as SCL:
   "AI_B4_Pct_RPC306_VFD" := SCALE_X(MIN := 20.0, VALUE := "Sim_Val_Norm", MAX := 80.0);
END_REGION

REGION Network 91: Tỷ lệ hóa AI_B4_Pres_FDF_mmWC (7.0 - 8.0 mmWC)
   RUNG wire#powerrail
      { S7_Templates := "[SrcType := Real, DestType := Real]" } Scale(min := 7.0, value := "Sim_Val_Norm", max := 8.0, out => "AI_B4_Pres_FDF_mmWC")
   END_RUNG
   // the same network as SCL:
   "AI_B4_Pres_FDF_mmWC" := SCALE_X(MIN := 7.0, VALUE := "Sim_Val_Norm", MAX := 8.0);
END_REGION

REGION Network 92: Tỷ lệ hóa AI_B4_TEST1_Value (0.0 - 100.0 )
   RUNG wire#powerrail
      { S7_Templates := "[SrcType := Real, DestType := Real]" } Scale(min := 0.0, value := "Sim_Val_Norm", max := 100.0, out => "AI_B4_TEST1_Value")
   END_RUNG
   // the same network as SCL:
   "AI_B4_TEST1_Value" := SCALE_X(MIN := 0.0, VALUE := "Sim_Val_Norm", MAX := 100.0);
END_REGION

REGION Network 93: Tỷ lệ hóa AI_B4_Pct_PAF1_SP (20.0 - 80.0 %)
   RUNG wire#powerrail
      { S7_Templates := "[SrcType := Real, DestType := Real]" } Scale(min := 20.0, value := "Sim_Val_Norm", max := 80.0, out => "AI_B4_Pct_PAF1_SP")
   END_RUNG
   // the same network as SCL:
   "AI_B4_Pct_PAF1_SP" := SCALE_X(MIN := 20.0, VALUE := "Sim_Val_Norm", MAX := 80.0);
END_REGION

REGION Network 94: Tỷ lệ hóa AI_B4_Pct_PAF1_PV (20.0 - 80.0 %)
   RUNG wire#powerrail
      { S7_Templates := "[SrcType := Real, DestType := Real]" } Scale(min := 20.0, value := "Sim_Val_Norm", max := 80.0, out => "AI_B4_Pct_PAF1_PV")
   END_RUNG
   // the same network as SCL:
   "AI_B4_Pct_PAF1_PV" := SCALE_X(MIN := 20.0, VALUE := "Sim_Val_Norm", MAX := 80.0);
END_REGION

REGION Network 95: Tỷ lệ hóa AI_B4_Pres_PAF2_mmWC (7.0 - 8.0 mmWC)
   RUNG wire#powerrail
      { S7_Templates := "[SrcType := Real, DestType := Real]" } Scale(min := 7.0, value := "Sim_Val_Norm", max := 8.0, out => "AI_B4_Pres_PAF2_mmWC")
   END_RUNG
   // the same network as SCL:
   "AI_B4_Pres_PAF2_mmWC" := SCALE_X(MIN := 7.0, VALUE := "Sim_Val_Norm", MAX := 8.0);
END_REGION

REGION Network 96: Tỷ lệ hóa AI_B4_RPM_PAF2 (800.0 - 1200.0 RPM)
   RUNG wire#powerrail
      { S7_Templates := "[SrcType := Real, DestType := Real]" } Scale(min := 800.0, value := "Sim_Val_Norm", max := 1200.0, out => "AI_B4_RPM_PAF2")
   END_RUNG
   // the same network as SCL:
   "AI_B4_RPM_PAF2" := SCALE_X(MIN := 800.0, VALUE := "Sim_Val_Norm", MAX := 1200.0);
END_REGION

REGION Network 97: Tỷ lệ hóa AI_B4_Pct_RPC308b_SP (20.0 - 80.0 %)
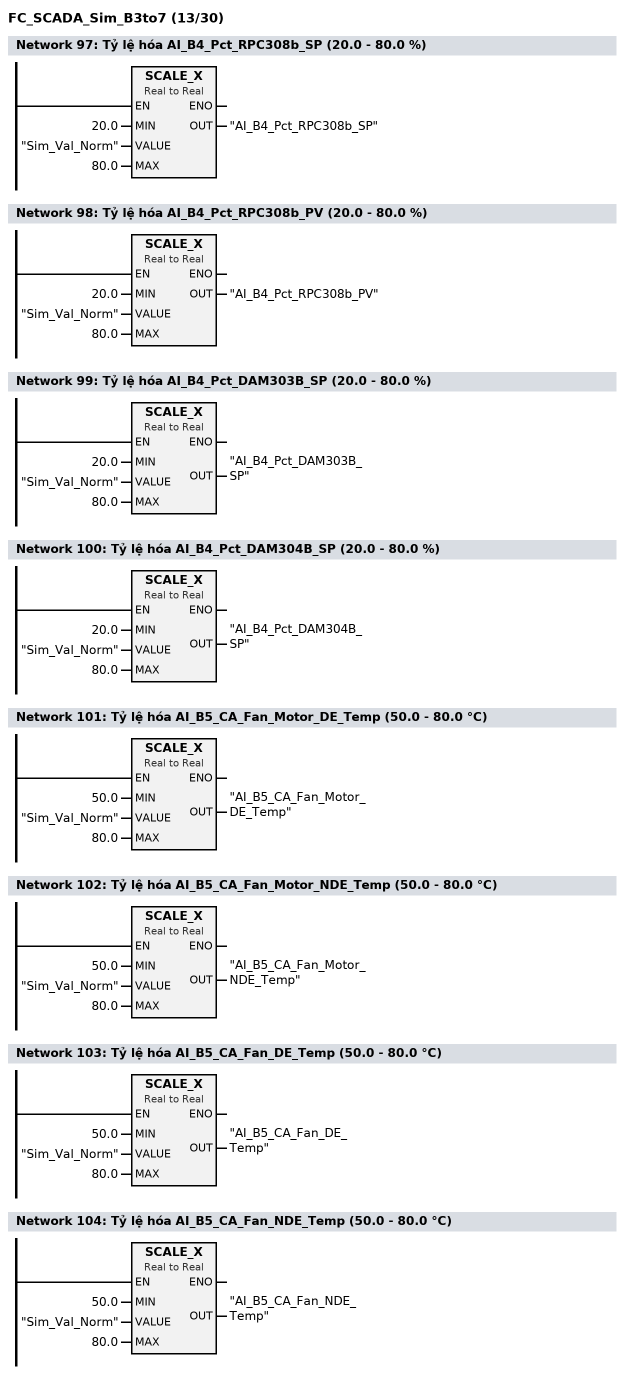
   RUNG wire#powerrail
      { S7_Templates := "[SrcType := Real, DestType := Real]" } Scale(min := 20.0, value := "Sim_Val_Norm", max := 80.0, out => "AI_B4_Pct_RPC308b_SP")
   END_RUNG
   // the same network as SCL:
   "AI_B4_Pct_RPC308b_SP" := SCALE_X(MIN := 20.0, VALUE := "Sim_Val_Norm", MAX := 80.0);
END_REGION

REGION Network 98: Tỷ lệ hóa AI_B4_Pct_RPC308b_PV (20.0 - 80.0 %)
   RUNG wire#powerrail
      { S7_Templates := "[SrcType := Real, DestType := Real]" } Scale(min := 20.0, value := "Sim_Val_Norm", max := 80.0, out => "AI_B4_Pct_RPC308b_PV")
   END_RUNG
   // the same network as SCL:
   "AI_B4_Pct_RPC308b_PV" := SCALE_X(MIN := 20.0, VALUE := "Sim_Val_Norm", MAX := 80.0);
END_REGION

REGION Network 99: Tỷ lệ hóa AI_B4_Pct_DAM303B_SP (20.0 - 80.0 %)
   RUNG wire#powerrail
      { S7_Templates := "[SrcType := Real, DestType := Real]" } Scale(min := 20.0, value := "Sim_Val_Norm", max := 80.0, out => "AI_B4_Pct_DAM303B_SP")
   END_RUNG
   // the same network as SCL:
   "AI_B4_Pct_DAM303B_SP" := SCALE_X(MIN := 20.0, VALUE := "Sim_Val_Norm", MAX := 80.0);
END_REGION

REGION Network 100: Tỷ lệ hóa AI_B4_Pct_DAM304B_SP (20.0 - 80.0 %)
   RUNG wire#powerrail
      { S7_Templates := "[SrcType := Real, DestType := Real]" } Scale(min := 20.0, value := "Sim_Val_Norm", max := 80.0, out => "AI_B4_Pct_DAM304B_SP")
   END_RUNG
   // the same network as SCL:
   "AI_B4_Pct_DAM304B_SP" := SCALE_X(MIN := 20.0, VALUE := "Sim_Val_Norm", MAX := 80.0);
END_REGION

REGION Network 101: Tỷ lệ hóa AI_B5_CA_Fan_Motor_DE_Temp (50.0 - 80.0 °C)
   RUNG wire#powerrail
      { S7_Templates := "[SrcType := Real, DestType := Real]" } Scale(min := 50.0, value := "Sim_Val_Norm", max := 80.0, out => "AI_B5_CA_Fan_Motor_DE_Temp")
   END_RUNG
   // the same network as SCL:
   "AI_B5_CA_Fan_Motor_DE_Temp" := SCALE_X(MIN := 50.0, VALUE := "Sim_Val_Norm", MAX := 80.0);
END_REGION

REGION Network 102: Tỷ lệ hóa AI_B5_CA_Fan_Motor_NDE_Temp (50.0 - 80.0 °C)
   RUNG wire#powerrail
      { S7_Templates := "[SrcType := Real, DestType := Real]" } Scale(min := 50.0, value := "Sim_Val_Norm", max := 80.0, out => "AI_B5_CA_Fan_Motor_NDE_Temp")
   END_RUNG
   // the same network as SCL:
   "AI_B5_CA_Fan_Motor_NDE_Temp" := SCALE_X(MIN := 50.0, VALUE := "Sim_Val_Norm", MAX := 80.0);
END_REGION

REGION Network 103: Tỷ lệ hóa AI_B5_CA_Fan_DE_Temp (50.0 - 80.0 °C)
   RUNG wire#powerrail
      { S7_Templates := "[SrcType := Real, DestType := Real]" } Scale(min := 50.0, value := "Sim_Val_Norm", max := 80.0, out => "AI_B5_CA_Fan_DE_Temp")
   END_RUNG
   // the same network as SCL:
   "AI_B5_CA_Fan_DE_Temp" := SCALE_X(MIN := 50.0, VALUE := "Sim_Val_Norm", MAX := 80.0);
END_REGION

REGION Network 104: Tỷ lệ hóa AI_B5_CA_Fan_NDE_Temp (50.0 - 80.0 °C)
   RUNG wire#powerrail
      { S7_Templates := "[SrcType := Real, DestType := Real]" } Scale(min := 50.0, value := "Sim_Val_Norm", max := 80.0, out => "AI_B5_CA_Fan_NDE_Temp")
   END_RUNG
   // the same network as SCL:
   "AI_B5_CA_Fan_NDE_Temp" := SCALE_X(MIN := 50.0, VALUE := "Sim_Val_Norm", MAX := 80.0);
END_REGION

REGION Network 105: Tỷ lệ hóa AI_B5_CA_Fan_DE_Vib (0.0 - 10.0 mm/s)
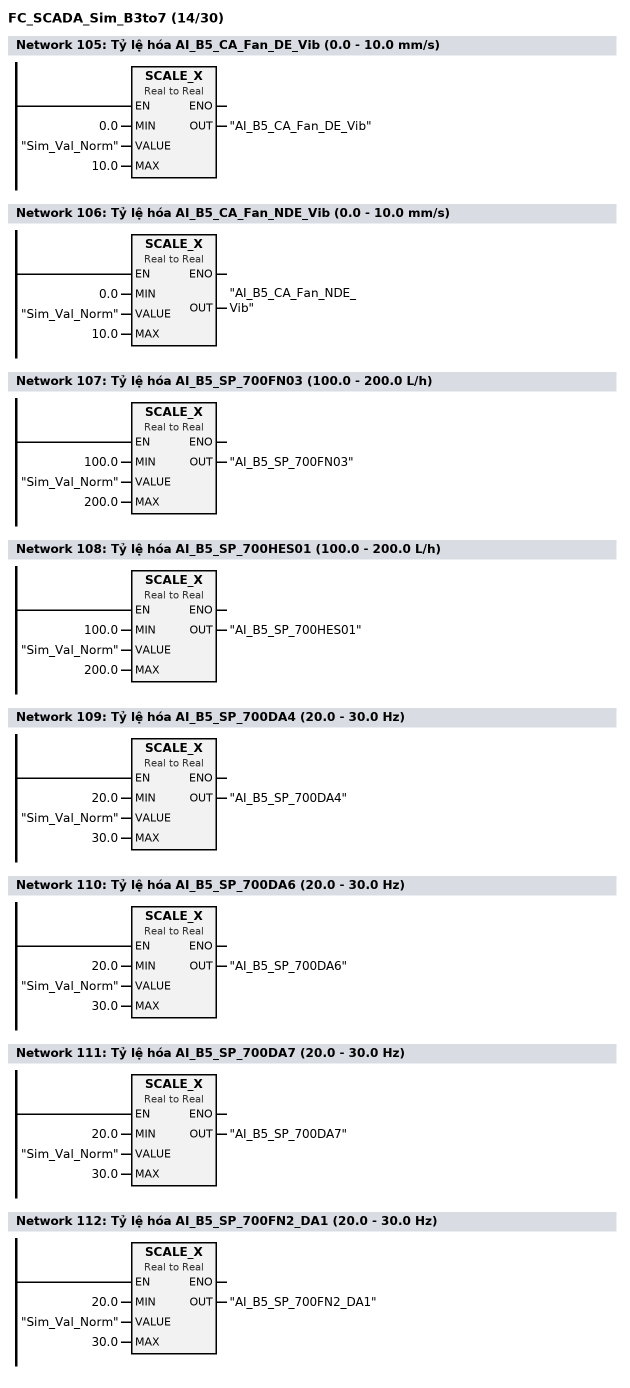
   RUNG wire#powerrail
      { S7_Templates := "[SrcType := Real, DestType := Real]" } Scale(min := 0.0, value := "Sim_Val_Norm", max := 10.0, out => "AI_B5_CA_Fan_DE_Vib")
   END_RUNG
   // the same network as SCL:
   "AI_B5_CA_Fan_DE_Vib" := SCALE_X(MIN := 0.0, VALUE := "Sim_Val_Norm", MAX := 10.0);
END_REGION

REGION Network 106: Tỷ lệ hóa AI_B5_CA_Fan_NDE_Vib (0.0 - 10.0 mm/s)
   RUNG wire#powerrail
      { S7_Templates := "[SrcType := Real, DestType := Real]" } Scale(min := 0.0, value := "Sim_Val_Norm", max := 10.0, out => "AI_B5_CA_Fan_NDE_Vib")
   END_RUNG
   // the same network as SCL:
   "AI_B5_CA_Fan_NDE_Vib" := SCALE_X(MIN := 0.0, VALUE := "Sim_Val_Norm", MAX := 10.0);
END_REGION

REGION Network 107: Tỷ lệ hóa AI_B5_SP_700FN03 (100.0 - 200.0 L/h)
   RUNG wire#powerrail
      { S7_Templates := "[SrcType := Real, DestType := Real]" } Scale(min := 100.0, value := "Sim_Val_Norm", max := 200.0, out => "AI_B5_SP_700FN03")
   END_RUNG
   // the same network as SCL:
   "AI_B5_SP_700FN03" := SCALE_X(MIN := 100.0, VALUE := "Sim_Val_Norm", MAX := 200.0);
END_REGION

REGION Network 108: Tỷ lệ hóa AI_B5_SP_700HES01 (100.0 - 200.0 L/h)
   RUNG wire#powerrail
      { S7_Templates := "[SrcType := Real, DestType := Real]" } Scale(min := 100.0, value := "Sim_Val_Norm", max := 200.0, out => "AI_B5_SP_700HES01")
   END_RUNG
   // the same network as SCL:
   "AI_B5_SP_700HES01" := SCALE_X(MIN := 100.0, VALUE := "Sim_Val_Norm", MAX := 200.0);
END_REGION

REGION Network 109: Tỷ lệ hóa AI_B5_SP_700DA4 (20.0 - 30.0 Hz)
   RUNG wire#powerrail
      { S7_Templates := "[SrcType := Real, DestType := Real]" } Scale(min := 20.0, value := "Sim_Val_Norm", max := 30.0, out => "AI_B5_SP_700DA4")
   END_RUNG
   // the same network as SCL:
   "AI_B5_SP_700DA4" := SCALE_X(MIN := 20.0, VALUE := "Sim_Val_Norm", MAX := 30.0);
END_REGION

REGION Network 110: Tỷ lệ hóa AI_B5_SP_700DA6 (20.0 - 30.0 Hz)
   RUNG wire#powerrail
      { S7_Templates := "[SrcType := Real, DestType := Real]" } Scale(min := 20.0, value := "Sim_Val_Norm", max := 30.0, out => "AI_B5_SP_700DA6")
   END_RUNG
   // the same network as SCL:
   "AI_B5_SP_700DA6" := SCALE_X(MIN := 20.0, VALUE := "Sim_Val_Norm", MAX := 30.0);
END_REGION

REGION Network 111: Tỷ lệ hóa AI_B5_SP_700DA7 (20.0 - 30.0 Hz)
   RUNG wire#powerrail
      { S7_Templates := "[SrcType := Real, DestType := Real]" } Scale(min := 20.0, value := "Sim_Val_Norm", max := 30.0, out => "AI_B5_SP_700DA7")
   END_RUNG
   // the same network as SCL:
   "AI_B5_SP_700DA7" := SCALE_X(MIN := 20.0, VALUE := "Sim_Val_Norm", MAX := 30.0);
END_REGION

REGION Network 112: Tỷ lệ hóa AI_B5_SP_700FN2_DA1 (20.0 - 30.0 Hz)
   RUNG wire#powerrail
      { S7_Templates := "[SrcType := Real, DestType := Real]" } Scale(min := 20.0, value := "Sim_Val_Norm", max := 30.0, out => "AI_B5_SP_700FN2_DA1")
   END_RUNG
   // the same network as SCL:
   "AI_B5_SP_700FN2_DA1" := SCALE_X(MIN := 20.0, VALUE := "Sim_Val_Norm", MAX := 30.0);
END_REGION

REGION Network 113: Tỷ lệ hóa AI_B5_Sep_Motor_Top_Temp (50.0 - 80.0 °C)
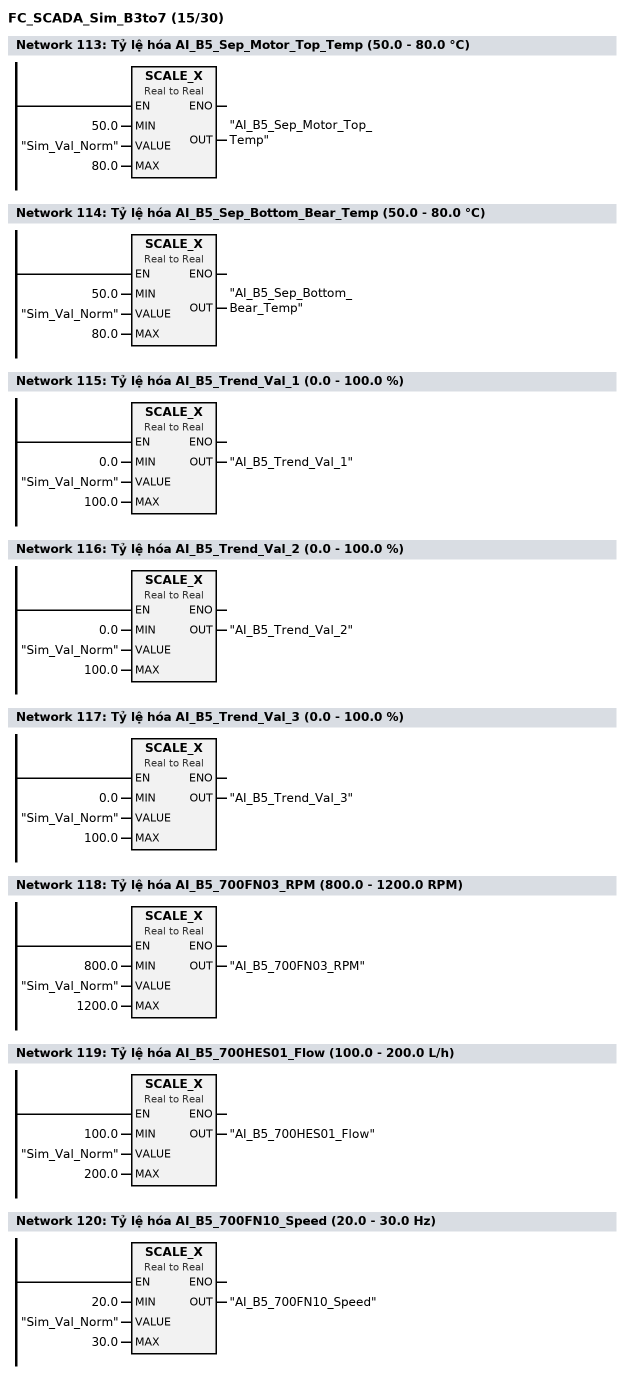
   RUNG wire#powerrail
      { S7_Templates := "[SrcType := Real, DestType := Real]" } Scale(min := 50.0, value := "Sim_Val_Norm", max := 80.0, out => "AI_B5_Sep_Motor_Top_Temp")
   END_RUNG
   // the same network as SCL:
   "AI_B5_Sep_Motor_Top_Temp" := SCALE_X(MIN := 50.0, VALUE := "Sim_Val_Norm", MAX := 80.0);
END_REGION

REGION Network 114: Tỷ lệ hóa AI_B5_Sep_Bottom_Bear_Temp (50.0 - 80.0 °C)
   RUNG wire#powerrail
      { S7_Templates := "[SrcType := Real, DestType := Real]" } Scale(min := 50.0, value := "Sim_Val_Norm", max := 80.0, out => "AI_B5_Sep_Bottom_Bear_Temp")
   END_RUNG
   // the same network as SCL:
   "AI_B5_Sep_Bottom_Bear_Temp" := SCALE_X(MIN := 50.0, VALUE := "Sim_Val_Norm", MAX := 80.0);
END_REGION

REGION Network 115: Tỷ lệ hóa AI_B5_Trend_Val_1 (0.0 - 100.0 %)
   RUNG wire#powerrail
      { S7_Templates := "[SrcType := Real, DestType := Real]" } Scale(min := 0.0, value := "Sim_Val_Norm", max := 100.0, out => "AI_B5_Trend_Val_1")
   END_RUNG
   // the same network as SCL:
   "AI_B5_Trend_Val_1" := SCALE_X(MIN := 0.0, VALUE := "Sim_Val_Norm", MAX := 100.0);
END_REGION

REGION Network 116: Tỷ lệ hóa AI_B5_Trend_Val_2 (0.0 - 100.0 %)
   RUNG wire#powerrail
      { S7_Templates := "[SrcType := Real, DestType := Real]" } Scale(min := 0.0, value := "Sim_Val_Norm", max := 100.0, out => "AI_B5_Trend_Val_2")
   END_RUNG
   // the same network as SCL:
   "AI_B5_Trend_Val_2" := SCALE_X(MIN := 0.0, VALUE := "Sim_Val_Norm", MAX := 100.0);
END_REGION

REGION Network 117: Tỷ lệ hóa AI_B5_Trend_Val_3 (0.0 - 100.0 %)
   RUNG wire#powerrail
      { S7_Templates := "[SrcType := Real, DestType := Real]" } Scale(min := 0.0, value := "Sim_Val_Norm", max := 100.0, out => "AI_B5_Trend_Val_3")
   END_RUNG
   // the same network as SCL:
   "AI_B5_Trend_Val_3" := SCALE_X(MIN := 0.0, VALUE := "Sim_Val_Norm", MAX := 100.0);
END_REGION

REGION Network 118: Tỷ lệ hóa AI_B5_700FN03_RPM (800.0 - 1200.0 RPM)
   RUNG wire#powerrail
      { S7_Templates := "[SrcType := Real, DestType := Real]" } Scale(min := 800.0, value := "Sim_Val_Norm", max := 1200.0, out => "AI_B5_700FN03_RPM")
   END_RUNG
   // the same network as SCL:
   "AI_B5_700FN03_RPM" := SCALE_X(MIN := 800.0, VALUE := "Sim_Val_Norm", MAX := 1200.0);
END_REGION

REGION Network 119: Tỷ lệ hóa AI_B5_700HES01_Flow (100.0 - 200.0 L/h)
   RUNG wire#powerrail
      { S7_Templates := "[SrcType := Real, DestType := Real]" } Scale(min := 100.0, value := "Sim_Val_Norm", max := 200.0, out => "AI_B5_700HES01_Flow")
   END_RUNG
   // the same network as SCL:
   "AI_B5_700HES01_Flow" := SCALE_X(MIN := 100.0, VALUE := "Sim_Val_Norm", MAX := 200.0);
END_REGION

REGION Network 120: Tỷ lệ hóa AI_B5_700FN10_Speed (20.0 - 30.0 Hz)
   RUNG wire#powerrail
      { S7_Templates := "[SrcType := Real, DestType := Real]" } Scale(min := 20.0, value := "Sim_Val_Norm", max := 30.0, out => "AI_B5_700FN10_Speed")
   END_RUNG
   // the same network as SCL:
   "AI_B5_700FN10_Speed" := SCALE_X(MIN := 20.0, VALUE := "Sim_Val_Norm", MAX := 30.0);
END_REGION

REGION Network 121: Tỷ lệ hóa AI_B5_700CM01_Current (50.0 - 200.0 A)
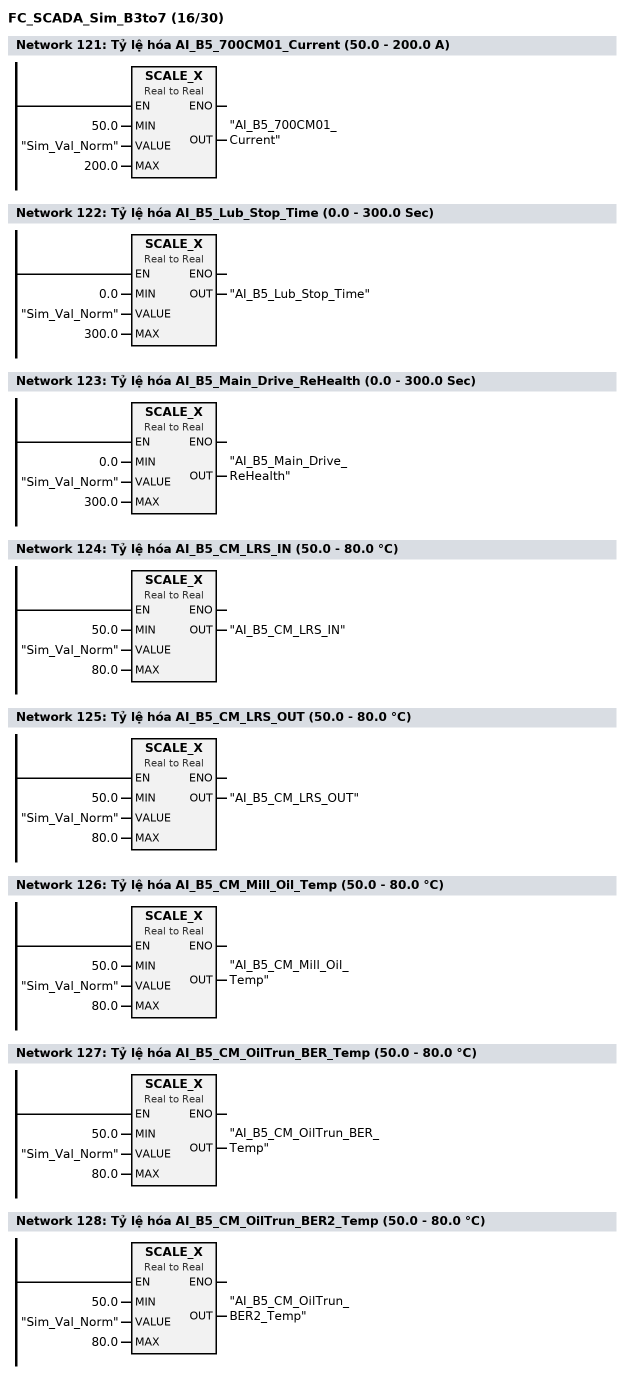
   RUNG wire#powerrail
      { S7_Templates := "[SrcType := Real, DestType := Real]" } Scale(min := 50.0, value := "Sim_Val_Norm", max := 200.0, out => "AI_B5_700CM01_Current")
   END_RUNG
   // the same network as SCL:
   "AI_B5_700CM01_Current" := SCALE_X(MIN := 50.0, VALUE := "Sim_Val_Norm", MAX := 200.0);
END_REGION

REGION Network 122: Tỷ lệ hóa AI_B5_Lub_Stop_Time (0.0 - 300.0 Sec)
   RUNG wire#powerrail
      { S7_Templates := "[SrcType := Real, DestType := Real]" } Scale(min := 0.0, value := "Sim_Val_Norm", max := 300.0, out => "AI_B5_Lub_Stop_Time")
   END_RUNG
   // the same network as SCL:
   "AI_B5_Lub_Stop_Time" := SCALE_X(MIN := 0.0, VALUE := "Sim_Val_Norm", MAX := 300.0);
END_REGION

REGION Network 123: Tỷ lệ hóa AI_B5_Main_Drive_ReHealth (0.0 - 300.0 Sec)
   RUNG wire#powerrail
      { S7_Templates := "[SrcType := Real, DestType := Real]" } Scale(min := 0.0, value := "Sim_Val_Norm", max := 300.0, out => "AI_B5_Main_Drive_ReHealth")
   END_RUNG
   // the same network as SCL:
   "AI_B5_Main_Drive_ReHealth" := SCALE_X(MIN := 0.0, VALUE := "Sim_Val_Norm", MAX := 300.0);
END_REGION

REGION Network 124: Tỷ lệ hóa AI_B5_CM_LRS_IN (50.0 - 80.0 °C)
   RUNG wire#powerrail
      { S7_Templates := "[SrcType := Real, DestType := Real]" } Scale(min := 50.0, value := "Sim_Val_Norm", max := 80.0, out => "AI_B5_CM_LRS_IN")
   END_RUNG
   // the same network as SCL:
   "AI_B5_CM_LRS_IN" := SCALE_X(MIN := 50.0, VALUE := "Sim_Val_Norm", MAX := 80.0);
END_REGION

REGION Network 125: Tỷ lệ hóa AI_B5_CM_LRS_OUT (50.0 - 80.0 °C)
   RUNG wire#powerrail
      { S7_Templates := "[SrcType := Real, DestType := Real]" } Scale(min := 50.0, value := "Sim_Val_Norm", max := 80.0, out => "AI_B5_CM_LRS_OUT")
   END_RUNG
   // the same network as SCL:
   "AI_B5_CM_LRS_OUT" := SCALE_X(MIN := 50.0, VALUE := "Sim_Val_Norm", MAX := 80.0);
END_REGION

REGION Network 126: Tỷ lệ hóa AI_B5_CM_Mill_Oil_Temp (50.0 - 80.0 °C)
   RUNG wire#powerrail
      { S7_Templates := "[SrcType := Real, DestType := Real]" } Scale(min := 50.0, value := "Sim_Val_Norm", max := 80.0, out => "AI_B5_CM_Mill_Oil_Temp")
   END_RUNG
   // the same network as SCL:
   "AI_B5_CM_Mill_Oil_Temp" := SCALE_X(MIN := 50.0, VALUE := "Sim_Val_Norm", MAX := 80.0);
END_REGION

REGION Network 127: Tỷ lệ hóa AI_B5_CM_OilTrun_BER_Temp (50.0 - 80.0 °C)
   RUNG wire#powerrail
      { S7_Templates := "[SrcType := Real, DestType := Real]" } Scale(min := 50.0, value := "Sim_Val_Norm", max := 80.0, out => "AI_B5_CM_OilTrun_BER_Temp")
   END_RUNG
   // the same network as SCL:
   "AI_B5_CM_OilTrun_BER_Temp" := SCALE_X(MIN := 50.0, VALUE := "Sim_Val_Norm", MAX := 80.0);
END_REGION

REGION Network 128: Tỷ lệ hóa AI_B5_CM_OilTrun_BER2_Temp (50.0 - 80.0 °C)
   RUNG wire#powerrail
      { S7_Templates := "[SrcType := Real, DestType := Real]" } Scale(min := 50.0, value := "Sim_Val_Norm", max := 80.0, out => "AI_B5_CM_OilTrun_BER2_Temp")
   END_RUNG
   // the same network as SCL:
   "AI_B5_CM_OilTrun_BER2_Temp" := SCALE_X(MIN := 50.0, VALUE := "Sim_Val_Norm", MAX := 80.0);
END_REGION

REGION Network 129: Tỷ lệ hóa AI_B5_CM_OilPinion_BER_Temp (50.0 - 80.0 °C)
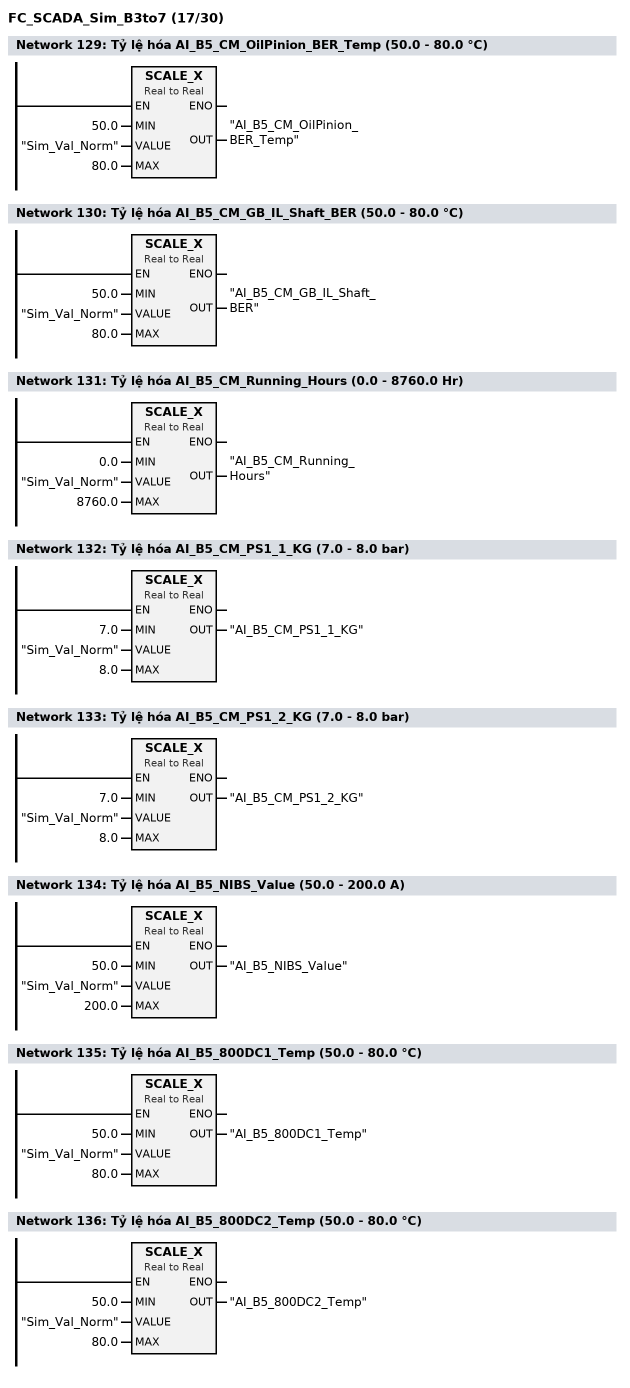
   RUNG wire#powerrail
      { S7_Templates := "[SrcType := Real, DestType := Real]" } Scale(min := 50.0, value := "Sim_Val_Norm", max := 80.0, out => "AI_B5_CM_OilPinion_BER_Temp")
   END_RUNG
   // the same network as SCL:
   "AI_B5_CM_OilPinion_BER_Temp" := SCALE_X(MIN := 50.0, VALUE := "Sim_Val_Norm", MAX := 80.0);
END_REGION

REGION Network 130: Tỷ lệ hóa AI_B5_CM_GB_IL_Shaft_BER (50.0 - 80.0 °C)
   RUNG wire#powerrail
      { S7_Templates := "[SrcType := Real, DestType := Real]" } Scale(min := 50.0, value := "Sim_Val_Norm", max := 80.0, out => "AI_B5_CM_GB_IL_Shaft_BER")
   END_RUNG
   // the same network as SCL:
   "AI_B5_CM_GB_IL_Shaft_BER" := SCALE_X(MIN := 50.0, VALUE := "Sim_Val_Norm", MAX := 80.0);
END_REGION

REGION Network 131: Tỷ lệ hóa AI_B5_CM_Running_Hours (0.0 - 8760.0 Hr)
   RUNG wire#powerrail
      { S7_Templates := "[SrcType := Real, DestType := Real]" } Scale(min := 0.0, value := "Sim_Val_Norm", max := 8760.0, out => "AI_B5_CM_Running_Hours")
   END_RUNG
   // the same network as SCL:
   "AI_B5_CM_Running_Hours" := SCALE_X(MIN := 0.0, VALUE := "Sim_Val_Norm", MAX := 8760.0);
END_REGION

REGION Network 132: Tỷ lệ hóa AI_B5_CM_PS1_1_KG (7.0 - 8.0 bar)
   RUNG wire#powerrail
      { S7_Templates := "[SrcType := Real, DestType := Real]" } Scale(min := 7.0, value := "Sim_Val_Norm", max := 8.0, out => "AI_B5_CM_PS1_1_KG")
   END_RUNG
   // the same network as SCL:
   "AI_B5_CM_PS1_1_KG" := SCALE_X(MIN := 7.0, VALUE := "Sim_Val_Norm", MAX := 8.0);
END_REGION

REGION Network 133: Tỷ lệ hóa AI_B5_CM_PS1_2_KG (7.0 - 8.0 bar)
   RUNG wire#powerrail
      { S7_Templates := "[SrcType := Real, DestType := Real]" } Scale(min := 7.0, value := "Sim_Val_Norm", max := 8.0, out => "AI_B5_CM_PS1_2_KG")
   END_RUNG
   // the same network as SCL:
   "AI_B5_CM_PS1_2_KG" := SCALE_X(MIN := 7.0, VALUE := "Sim_Val_Norm", MAX := 8.0);
END_REGION

REGION Network 134: Tỷ lệ hóa AI_B5_NIBS_Value (50.0 - 200.0 A)
   RUNG wire#powerrail
      { S7_Templates := "[SrcType := Real, DestType := Real]" } Scale(min := 50.0, value := "Sim_Val_Norm", max := 200.0, out => "AI_B5_NIBS_Value")
   END_RUNG
   // the same network as SCL:
   "AI_B5_NIBS_Value" := SCALE_X(MIN := 50.0, VALUE := "Sim_Val_Norm", MAX := 200.0);
END_REGION

REGION Network 135: Tỷ lệ hóa AI_B5_800DC1_Temp (50.0 - 80.0 °C)
   RUNG wire#powerrail
      { S7_Templates := "[SrcType := Real, DestType := Real]" } Scale(min := 50.0, value := "Sim_Val_Norm", max := 80.0, out => "AI_B5_800DC1_Temp")
   END_RUNG
   // the same network as SCL:
   "AI_B5_800DC1_Temp" := SCALE_X(MIN := 50.0, VALUE := "Sim_Val_Norm", MAX := 80.0);
END_REGION

REGION Network 136: Tỷ lệ hóa AI_B5_800DC2_Temp (50.0 - 80.0 °C)
   RUNG wire#powerrail
      { S7_Templates := "[SrcType := Real, DestType := Real]" } Scale(min := 50.0, value := "Sim_Val_Norm", max := 80.0, out => "AI_B5_800DC2_Temp")
   END_RUNG
   // the same network as SCL:
   "AI_B5_800DC2_Temp" := SCALE_X(MIN := 50.0, VALUE := "Sim_Val_Norm", MAX := 80.0);
END_REGION

REGION Network 137: Tỷ lệ hóa AI_B5_800FN1_Speed (20.0 - 30.0 Hz)
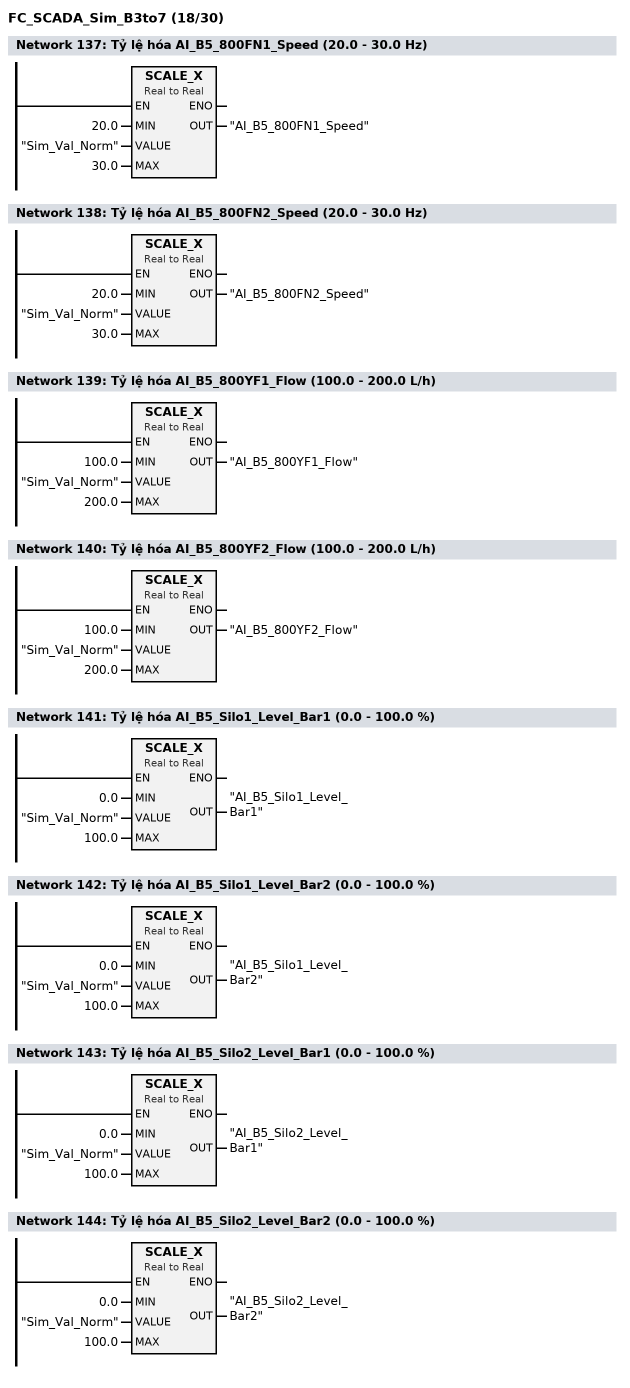
   RUNG wire#powerrail
      { S7_Templates := "[SrcType := Real, DestType := Real]" } Scale(min := 20.0, value := "Sim_Val_Norm", max := 30.0, out => "AI_B5_800FN1_Speed")
   END_RUNG
   // the same network as SCL:
   "AI_B5_800FN1_Speed" := SCALE_X(MIN := 20.0, VALUE := "Sim_Val_Norm", MAX := 30.0);
END_REGION

REGION Network 138: Tỷ lệ hóa AI_B5_800FN2_Speed (20.0 - 30.0 Hz)
   RUNG wire#powerrail
      { S7_Templates := "[SrcType := Real, DestType := Real]" } Scale(min := 20.0, value := "Sim_Val_Norm", max := 30.0, out => "AI_B5_800FN2_Speed")
   END_RUNG
   // the same network as SCL:
   "AI_B5_800FN2_Speed" := SCALE_X(MIN := 20.0, VALUE := "Sim_Val_Norm", MAX := 30.0);
END_REGION

REGION Network 139: Tỷ lệ hóa AI_B5_800YF1_Flow (100.0 - 200.0 L/h)
   RUNG wire#powerrail
      { S7_Templates := "[SrcType := Real, DestType := Real]" } Scale(min := 100.0, value := "Sim_Val_Norm", max := 200.0, out => "AI_B5_800YF1_Flow")
   END_RUNG
   // the same network as SCL:
   "AI_B5_800YF1_Flow" := SCALE_X(MIN := 100.0, VALUE := "Sim_Val_Norm", MAX := 200.0);
END_REGION

REGION Network 140: Tỷ lệ hóa AI_B5_800YF2_Flow (100.0 - 200.0 L/h)
   RUNG wire#powerrail
      { S7_Templates := "[SrcType := Real, DestType := Real]" } Scale(min := 100.0, value := "Sim_Val_Norm", max := 200.0, out => "AI_B5_800YF2_Flow")
   END_RUNG
   // the same network as SCL:
   "AI_B5_800YF2_Flow" := SCALE_X(MIN := 100.0, VALUE := "Sim_Val_Norm", MAX := 200.0);
END_REGION

REGION Network 141: Tỷ lệ hóa AI_B5_Silo1_Level_Bar1 (0.0 - 100.0 %)
   RUNG wire#powerrail
      { S7_Templates := "[SrcType := Real, DestType := Real]" } Scale(min := 0.0, value := "Sim_Val_Norm", max := 100.0, out => "AI_B5_Silo1_Level_Bar1")
   END_RUNG
   // the same network as SCL:
   "AI_B5_Silo1_Level_Bar1" := SCALE_X(MIN := 0.0, VALUE := "Sim_Val_Norm", MAX := 100.0);
END_REGION

REGION Network 142: Tỷ lệ hóa AI_B5_Silo1_Level_Bar2 (0.0 - 100.0 %)
   RUNG wire#powerrail
      { S7_Templates := "[SrcType := Real, DestType := Real]" } Scale(min := 0.0, value := "Sim_Val_Norm", max := 100.0, out => "AI_B5_Silo1_Level_Bar2")
   END_RUNG
   // the same network as SCL:
   "AI_B5_Silo1_Level_Bar2" := SCALE_X(MIN := 0.0, VALUE := "Sim_Val_Norm", MAX := 100.0);
END_REGION

REGION Network 143: Tỷ lệ hóa AI_B5_Silo2_Level_Bar1 (0.0 - 100.0 %)
   RUNG wire#powerrail
      { S7_Templates := "[SrcType := Real, DestType := Real]" } Scale(min := 0.0, value := "Sim_Val_Norm", max := 100.0, out => "AI_B5_Silo2_Level_Bar1")
   END_RUNG
   // the same network as SCL:
   "AI_B5_Silo2_Level_Bar1" := SCALE_X(MIN := 0.0, VALUE := "Sim_Val_Norm", MAX := 100.0);
END_REGION

REGION Network 144: Tỷ lệ hóa AI_B5_Silo2_Level_Bar2 (0.0 - 100.0 %)
   RUNG wire#powerrail
      { S7_Templates := "[SrcType := Real, DestType := Real]" } Scale(min := 0.0, value := "Sim_Val_Norm", max := 100.0, out => "AI_B5_Silo2_Level_Bar2")
   END_RUNG
   // the same network as SCL:
   "AI_B5_Silo2_Level_Bar2" := SCALE_X(MIN := 0.0, VALUE := "Sim_Val_Norm", MAX := 100.0);
END_REGION

REGION Network 145: Tỷ lệ hóa AI_B5_700FN01_Speed (20.0 - 30.0 Hz)
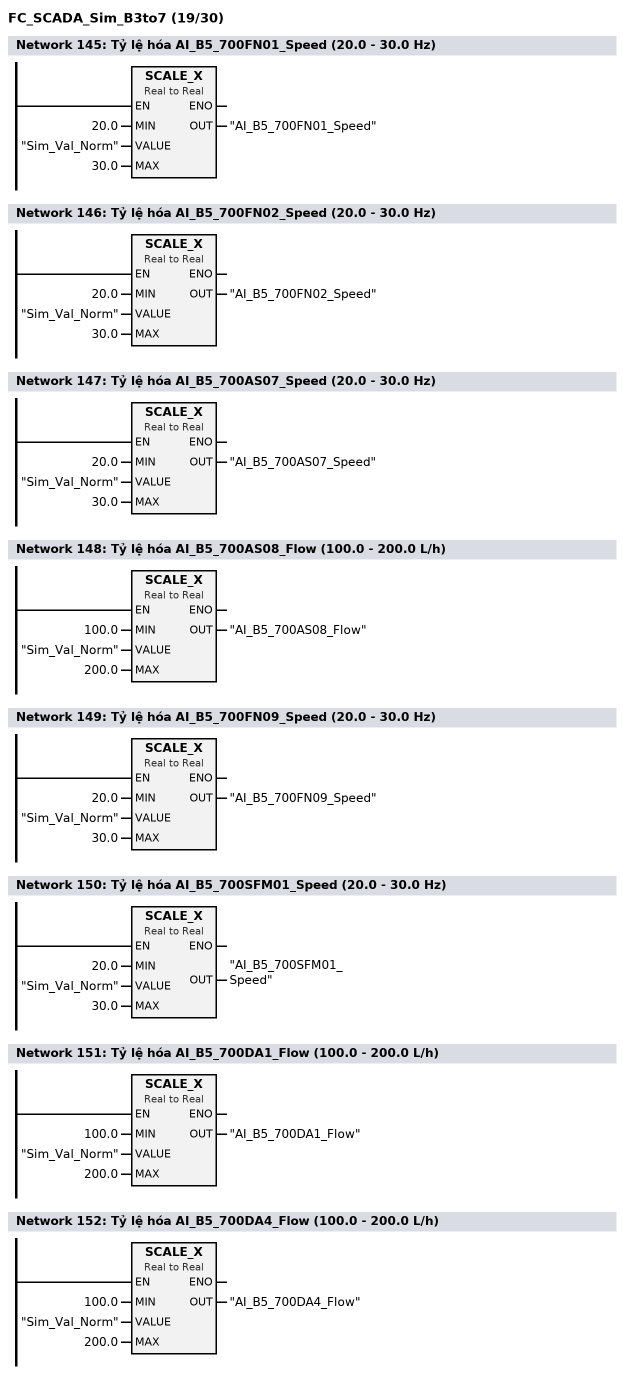
   RUNG wire#powerrail
      { S7_Templates := "[SrcType := Real, DestType := Real]" } Scale(min := 20.0, value := "Sim_Val_Norm", max := 30.0, out => "AI_B5_700FN01_Speed")
   END_RUNG
   // the same network as SCL:
   "AI_B5_700FN01_Speed" := SCALE_X(MIN := 20.0, VALUE := "Sim_Val_Norm", MAX := 30.0);
END_REGION

REGION Network 146: Tỷ lệ hóa AI_B5_700FN02_Speed (20.0 - 30.0 Hz)
   RUNG wire#powerrail
      { S7_Templates := "[SrcType := Real, DestType := Real]" } Scale(min := 20.0, value := "Sim_Val_Norm", max := 30.0, out => "AI_B5_700FN02_Speed")
   END_RUNG
   // the same network as SCL:
   "AI_B5_700FN02_Speed" := SCALE_X(MIN := 20.0, VALUE := "Sim_Val_Norm", MAX := 30.0);
END_REGION

REGION Network 147: Tỷ lệ hóa AI_B5_700AS07_Speed (20.0 - 30.0 Hz)
   RUNG wire#powerrail
      { S7_Templates := "[SrcType := Real, DestType := Real]" } Scale(min := 20.0, value := "Sim_Val_Norm", max := 30.0, out => "AI_B5_700AS07_Speed")
   END_RUNG
   // the same network as SCL:
   "AI_B5_700AS07_Speed" := SCALE_X(MIN := 20.0, VALUE := "Sim_Val_Norm", MAX := 30.0);
END_REGION

REGION Network 148: Tỷ lệ hóa AI_B5_700AS08_Flow (100.0 - 200.0 L/h)
   RUNG wire#powerrail
      { S7_Templates := "[SrcType := Real, DestType := Real]" } Scale(min := 100.0, value := "Sim_Val_Norm", max := 200.0, out => "AI_B5_700AS08_Flow")
   END_RUNG
   // the same network as SCL:
   "AI_B5_700AS08_Flow" := SCALE_X(MIN := 100.0, VALUE := "Sim_Val_Norm", MAX := 200.0);
END_REGION

REGION Network 149: Tỷ lệ hóa AI_B5_700FN09_Speed (20.0 - 30.0 Hz)
   RUNG wire#powerrail
      { S7_Templates := "[SrcType := Real, DestType := Real]" } Scale(min := 20.0, value := "Sim_Val_Norm", max := 30.0, out => "AI_B5_700FN09_Speed")
   END_RUNG
   // the same network as SCL:
   "AI_B5_700FN09_Speed" := SCALE_X(MIN := 20.0, VALUE := "Sim_Val_Norm", MAX := 30.0);
END_REGION

REGION Network 150: Tỷ lệ hóa AI_B5_700SFM01_Speed (20.0 - 30.0 Hz)
   RUNG wire#powerrail
      { S7_Templates := "[SrcType := Real, DestType := Real]" } Scale(min := 20.0, value := "Sim_Val_Norm", max := 30.0, out => "AI_B5_700SFM01_Speed")
   END_RUNG
   // the same network as SCL:
   "AI_B5_700SFM01_Speed" := SCALE_X(MIN := 20.0, VALUE := "Sim_Val_Norm", MAX := 30.0);
END_REGION

REGION Network 151: Tỷ lệ hóa AI_B5_700DA1_Flow (100.0 - 200.0 L/h)
   RUNG wire#powerrail
      { S7_Templates := "[SrcType := Real, DestType := Real]" } Scale(min := 100.0, value := "Sim_Val_Norm", max := 200.0, out => "AI_B5_700DA1_Flow")
   END_RUNG
   // the same network as SCL:
   "AI_B5_700DA1_Flow" := SCALE_X(MIN := 100.0, VALUE := "Sim_Val_Norm", MAX := 200.0);
END_REGION

REGION Network 152: Tỷ lệ hóa AI_B5_700DA4_Flow (100.0 - 200.0 L/h)
   RUNG wire#powerrail
      { S7_Templates := "[SrcType := Real, DestType := Real]" } Scale(min := 100.0, value := "Sim_Val_Norm", max := 200.0, out => "AI_B5_700DA4_Flow")
   END_RUNG
   // the same network as SCL:
   "AI_B5_700DA4_Flow" := SCALE_X(MIN := 100.0, VALUE := "Sim_Val_Norm", MAX := 200.0);
END_REGION

REGION Network 153: Tỷ lệ hóa AI_B5_700DA6_Temp (50.0 - 80.0 °C)
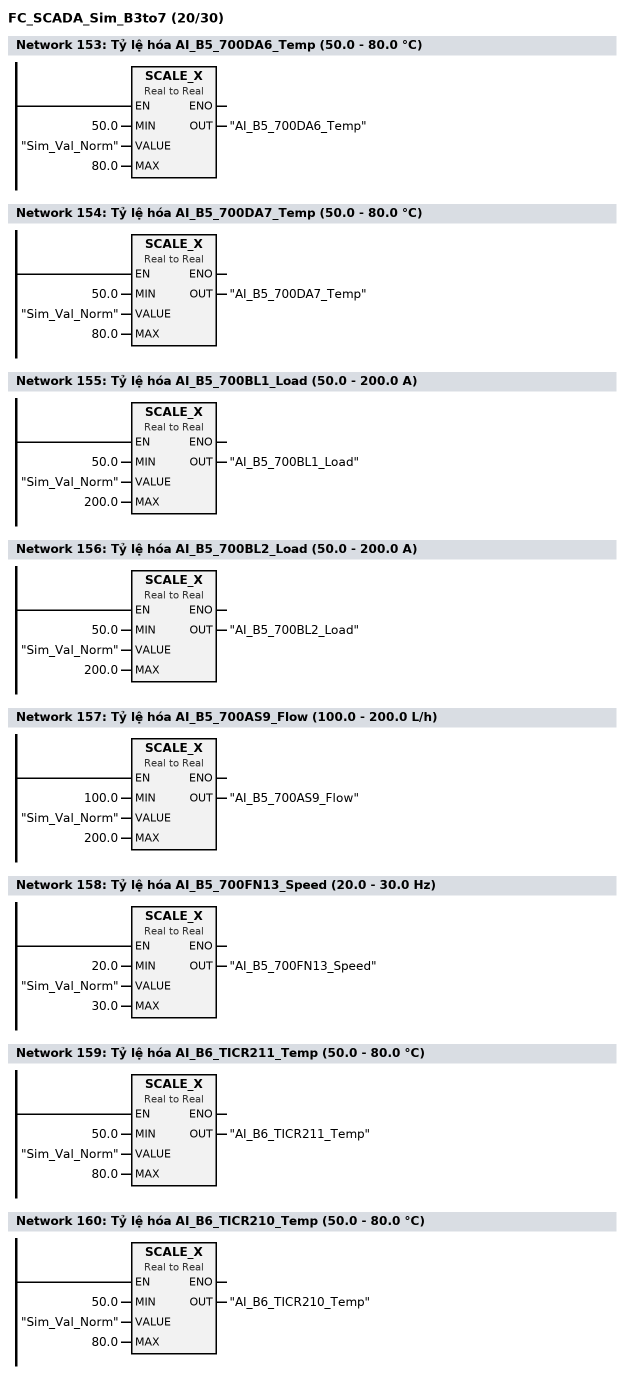
   RUNG wire#powerrail
      { S7_Templates := "[SrcType := Real, DestType := Real]" } Scale(min := 50.0, value := "Sim_Val_Norm", max := 80.0, out => "AI_B5_700DA6_Temp")
   END_RUNG
   // the same network as SCL:
   "AI_B5_700DA6_Temp" := SCALE_X(MIN := 50.0, VALUE := "Sim_Val_Norm", MAX := 80.0);
END_REGION

REGION Network 154: Tỷ lệ hóa AI_B5_700DA7_Temp (50.0 - 80.0 °C)
   RUNG wire#powerrail
      { S7_Templates := "[SrcType := Real, DestType := Real]" } Scale(min := 50.0, value := "Sim_Val_Norm", max := 80.0, out => "AI_B5_700DA7_Temp")
   END_RUNG
   // the same network as SCL:
   "AI_B5_700DA7_Temp" := SCALE_X(MIN := 50.0, VALUE := "Sim_Val_Norm", MAX := 80.0);
END_REGION

REGION Network 155: Tỷ lệ hóa AI_B5_700BL1_Load (50.0 - 200.0 A)
   RUNG wire#powerrail
      { S7_Templates := "[SrcType := Real, DestType := Real]" } Scale(min := 50.0, value := "Sim_Val_Norm", max := 200.0, out => "AI_B5_700BL1_Load")
   END_RUNG
   // the same network as SCL:
   "AI_B5_700BL1_Load" := SCALE_X(MIN := 50.0, VALUE := "Sim_Val_Norm", MAX := 200.0);
END_REGION

REGION Network 156: Tỷ lệ hóa AI_B5_700BL2_Load (50.0 - 200.0 A)
   RUNG wire#powerrail
      { S7_Templates := "[SrcType := Real, DestType := Real]" } Scale(min := 50.0, value := "Sim_Val_Norm", max := 200.0, out => "AI_B5_700BL2_Load")
   END_RUNG
   // the same network as SCL:
   "AI_B5_700BL2_Load" := SCALE_X(MIN := 50.0, VALUE := "Sim_Val_Norm", MAX := 200.0);
END_REGION

REGION Network 157: Tỷ lệ hóa AI_B5_700AS9_Flow (100.0 - 200.0 L/h)
   RUNG wire#powerrail
      { S7_Templates := "[SrcType := Real, DestType := Real]" } Scale(min := 100.0, value := "Sim_Val_Norm", max := 200.0, out => "AI_B5_700AS9_Flow")
   END_RUNG
   // the same network as SCL:
   "AI_B5_700AS9_Flow" := SCALE_X(MIN := 100.0, VALUE := "Sim_Val_Norm", MAX := 200.0);
END_REGION

REGION Network 158: Tỷ lệ hóa AI_B5_700FN13_Speed (20.0 - 30.0 Hz)
   RUNG wire#powerrail
      { S7_Templates := "[SrcType := Real, DestType := Real]" } Scale(min := 20.0, value := "Sim_Val_Norm", max := 30.0, out => "AI_B5_700FN13_Speed")
   END_RUNG
   // the same network as SCL:
   "AI_B5_700FN13_Speed" := SCALE_X(MIN := 20.0, VALUE := "Sim_Val_Norm", MAX := 30.0);
END_REGION

REGION Network 159: Tỷ lệ hóa AI_B6_TICR211_Temp (50.0 - 80.0 °C)
   RUNG wire#powerrail
      { S7_Templates := "[SrcType := Real, DestType := Real]" } Scale(min := 50.0, value := "Sim_Val_Norm", max := 80.0, out => "AI_B6_TICR211_Temp")
   END_RUNG
   // the same network as SCL:
   "AI_B6_TICR211_Temp" := SCALE_X(MIN := 50.0, VALUE := "Sim_Val_Norm", MAX := 80.0);
END_REGION

REGION Network 160: Tỷ lệ hóa AI_B6_TICR210_Temp (50.0 - 80.0 °C)
   RUNG wire#powerrail
      { S7_Templates := "[SrcType := Real, DestType := Real]" } Scale(min := 50.0, value := "Sim_Val_Norm", max := 80.0, out => "AI_B6_TICR210_Temp")
   END_RUNG
   // the same network as SCL:
   "AI_B6_TICR210_Temp" := SCALE_X(MIN := 50.0, VALUE := "Sim_Val_Norm", MAX := 80.0);
END_REGION

REGION Network 161: Tỷ lệ hóa AI_B6_TICR201_Tank_Temp (50.0 - 80.0 °C)
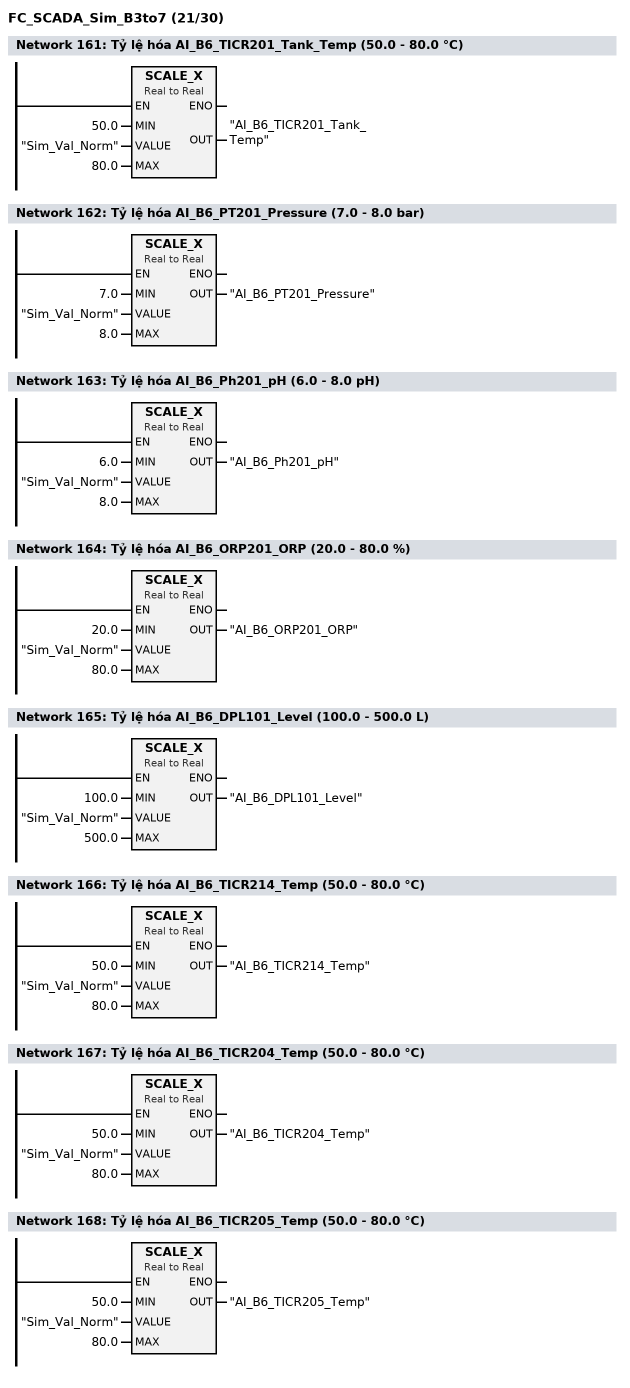
   RUNG wire#powerrail
      { S7_Templates := "[SrcType := Real, DestType := Real]" } Scale(min := 50.0, value := "Sim_Val_Norm", max := 80.0, out => "AI_B6_TICR201_Tank_Temp")
   END_RUNG
   // the same network as SCL:
   "AI_B6_TICR201_Tank_Temp" := SCALE_X(MIN := 50.0, VALUE := "Sim_Val_Norm", MAX := 80.0);
END_REGION

REGION Network 162: Tỷ lệ hóa AI_B6_PT201_Pressure (7.0 - 8.0 bar)
   RUNG wire#powerrail
      { S7_Templates := "[SrcType := Real, DestType := Real]" } Scale(min := 7.0, value := "Sim_Val_Norm", max := 8.0, out => "AI_B6_PT201_Pressure")
   END_RUNG
   // the same network as SCL:
   "AI_B6_PT201_Pressure" := SCALE_X(MIN := 7.0, VALUE := "Sim_Val_Norm", MAX := 8.0);
END_REGION

REGION Network 163: Tỷ lệ hóa AI_B6_Ph201_pH (6.0 - 8.0 pH)
   RUNG wire#powerrail
      { S7_Templates := "[SrcType := Real, DestType := Real]" } Scale(min := 6.0, value := "Sim_Val_Norm", max := 8.0, out => "AI_B6_Ph201_pH")
   END_RUNG
   // the same network as SCL:
   "AI_B6_Ph201_pH" := SCALE_X(MIN := 6.0, VALUE := "Sim_Val_Norm", MAX := 8.0);
END_REGION

REGION Network 164: Tỷ lệ hóa AI_B6_ORP201_ORP (20.0 - 80.0 %)
   RUNG wire#powerrail
      { S7_Templates := "[SrcType := Real, DestType := Real]" } Scale(min := 20.0, value := "Sim_Val_Norm", max := 80.0, out => "AI_B6_ORP201_ORP")
   END_RUNG
   // the same network as SCL:
   "AI_B6_ORP201_ORP" := SCALE_X(MIN := 20.0, VALUE := "Sim_Val_Norm", MAX := 80.0);
END_REGION

REGION Network 165: Tỷ lệ hóa AI_B6_DPL101_Level (100.0 - 500.0 L)
   RUNG wire#powerrail
      { S7_Templates := "[SrcType := Real, DestType := Real]" } Scale(min := 100.0, value := "Sim_Val_Norm", max := 500.0, out => "AI_B6_DPL101_Level")
   END_RUNG
   // the same network as SCL:
   "AI_B6_DPL101_Level" := SCALE_X(MIN := 100.0, VALUE := "Sim_Val_Norm", MAX := 500.0);
END_REGION

REGION Network 166: Tỷ lệ hóa AI_B6_TICR214_Temp (50.0 - 80.0 °C)
   RUNG wire#powerrail
      { S7_Templates := "[SrcType := Real, DestType := Real]" } Scale(min := 50.0, value := "Sim_Val_Norm", max := 80.0, out => "AI_B6_TICR214_Temp")
   END_RUNG
   // the same network as SCL:
   "AI_B6_TICR214_Temp" := SCALE_X(MIN := 50.0, VALUE := "Sim_Val_Norm", MAX := 80.0);
END_REGION

REGION Network 167: Tỷ lệ hóa AI_B6_TICR204_Temp (50.0 - 80.0 °C)
   RUNG wire#powerrail
      { S7_Templates := "[SrcType := Real, DestType := Real]" } Scale(min := 50.0, value := "Sim_Val_Norm", max := 80.0, out => "AI_B6_TICR204_Temp")
   END_RUNG
   // the same network as SCL:
   "AI_B6_TICR204_Temp" := SCALE_X(MIN := 50.0, VALUE := "Sim_Val_Norm", MAX := 80.0);
END_REGION

REGION Network 168: Tỷ lệ hóa AI_B6_TICR205_Temp (50.0 - 80.0 °C)
   RUNG wire#powerrail
      { S7_Templates := "[SrcType := Real, DestType := Real]" } Scale(min := 50.0, value := "Sim_Val_Norm", max := 80.0, out => "AI_B6_TICR205_Temp")
   END_RUNG
   // the same network as SCL:
   "AI_B6_TICR205_Temp" := SCALE_X(MIN := 50.0, VALUE := "Sim_Val_Norm", MAX := 80.0);
END_REGION

REGION Network 169: Tỷ lệ hóa AI_B6_TICR206_Temp (50.0 - 80.0 °C)
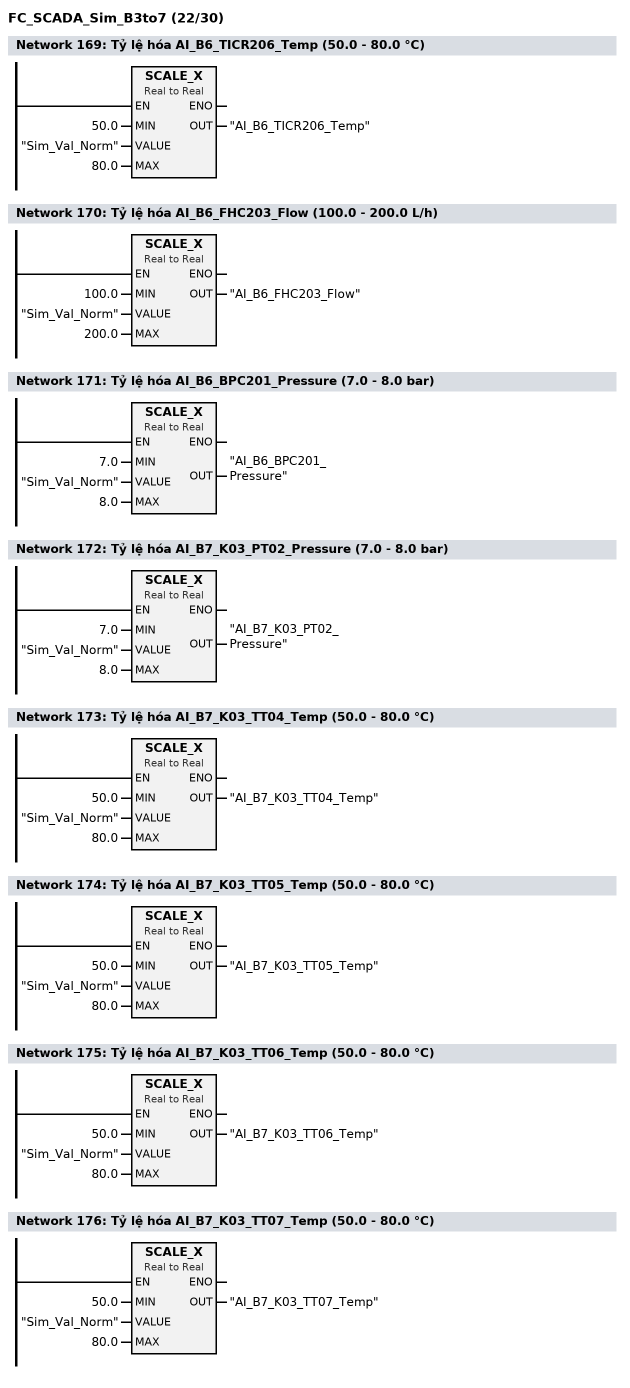
   RUNG wire#powerrail
      { S7_Templates := "[SrcType := Real, DestType := Real]" } Scale(min := 50.0, value := "Sim_Val_Norm", max := 80.0, out => "AI_B6_TICR206_Temp")
   END_RUNG
   // the same network as SCL:
   "AI_B6_TICR206_Temp" := SCALE_X(MIN := 50.0, VALUE := "Sim_Val_Norm", MAX := 80.0);
END_REGION

REGION Network 170: Tỷ lệ hóa AI_B6_FHC203_Flow (100.0 - 200.0 L/h)
   RUNG wire#powerrail
      { S7_Templates := "[SrcType := Real, DestType := Real]" } Scale(min := 100.0, value := "Sim_Val_Norm", max := 200.0, out => "AI_B6_FHC203_Flow")
   END_RUNG
   // the same network as SCL:
   "AI_B6_FHC203_Flow" := SCALE_X(MIN := 100.0, VALUE := "Sim_Val_Norm", MAX := 200.0);
END_REGION

REGION Network 171: Tỷ lệ hóa AI_B6_BPC201_Pressure (7.0 - 8.0 bar)
   RUNG wire#powerrail
      { S7_Templates := "[SrcType := Real, DestType := Real]" } Scale(min := 7.0, value := "Sim_Val_Norm", max := 8.0, out => "AI_B6_BPC201_Pressure")
   END_RUNG
   // the same network as SCL:
   "AI_B6_BPC201_Pressure" := SCALE_X(MIN := 7.0, VALUE := "Sim_Val_Norm", MAX := 8.0);
END_REGION

REGION Network 172: Tỷ lệ hóa AI_B7_K03_PT02_Pressure (7.0 - 8.0 bar)
   RUNG wire#powerrail
      { S7_Templates := "[SrcType := Real, DestType := Real]" } Scale(min := 7.0, value := "Sim_Val_Norm", max := 8.0, out => "AI_B7_K03_PT02_Pressure")
   END_RUNG
   // the same network as SCL:
   "AI_B7_K03_PT02_Pressure" := SCALE_X(MIN := 7.0, VALUE := "Sim_Val_Norm", MAX := 8.0);
END_REGION

REGION Network 173: Tỷ lệ hóa AI_B7_K03_TT04_Temp (50.0 - 80.0 °C)
   RUNG wire#powerrail
      { S7_Templates := "[SrcType := Real, DestType := Real]" } Scale(min := 50.0, value := "Sim_Val_Norm", max := 80.0, out => "AI_B7_K03_TT04_Temp")
   END_RUNG
   // the same network as SCL:
   "AI_B7_K03_TT04_Temp" := SCALE_X(MIN := 50.0, VALUE := "Sim_Val_Norm", MAX := 80.0);
END_REGION

REGION Network 174: Tỷ lệ hóa AI_B7_K03_TT05_Temp (50.0 - 80.0 °C)
   RUNG wire#powerrail
      { S7_Templates := "[SrcType := Real, DestType := Real]" } Scale(min := 50.0, value := "Sim_Val_Norm", max := 80.0, out => "AI_B7_K03_TT05_Temp")
   END_RUNG
   // the same network as SCL:
   "AI_B7_K03_TT05_Temp" := SCALE_X(MIN := 50.0, VALUE := "Sim_Val_Norm", MAX := 80.0);
END_REGION

REGION Network 175: Tỷ lệ hóa AI_B7_K03_TT06_Temp (50.0 - 80.0 °C)
   RUNG wire#powerrail
      { S7_Templates := "[SrcType := Real, DestType := Real]" } Scale(min := 50.0, value := "Sim_Val_Norm", max := 80.0, out => "AI_B7_K03_TT06_Temp")
   END_RUNG
   // the same network as SCL:
   "AI_B7_K03_TT06_Temp" := SCALE_X(MIN := 50.0, VALUE := "Sim_Val_Norm", MAX := 80.0);
END_REGION

REGION Network 176: Tỷ lệ hóa AI_B7_K03_TT07_Temp (50.0 - 80.0 °C)
   RUNG wire#powerrail
      { S7_Templates := "[SrcType := Real, DestType := Real]" } Scale(min := 50.0, value := "Sim_Val_Norm", max := 80.0, out => "AI_B7_K03_TT07_Temp")
   END_RUNG
   // the same network as SCL:
   "AI_B7_K03_TT07_Temp" := SCALE_X(MIN := 50.0, VALUE := "Sim_Val_Norm", MAX := 80.0);
END_REGION

REGION Network 177: Tỷ lệ hóa AI_B7_K03_PT07_Pressure (7.0 - 8.0 bar)
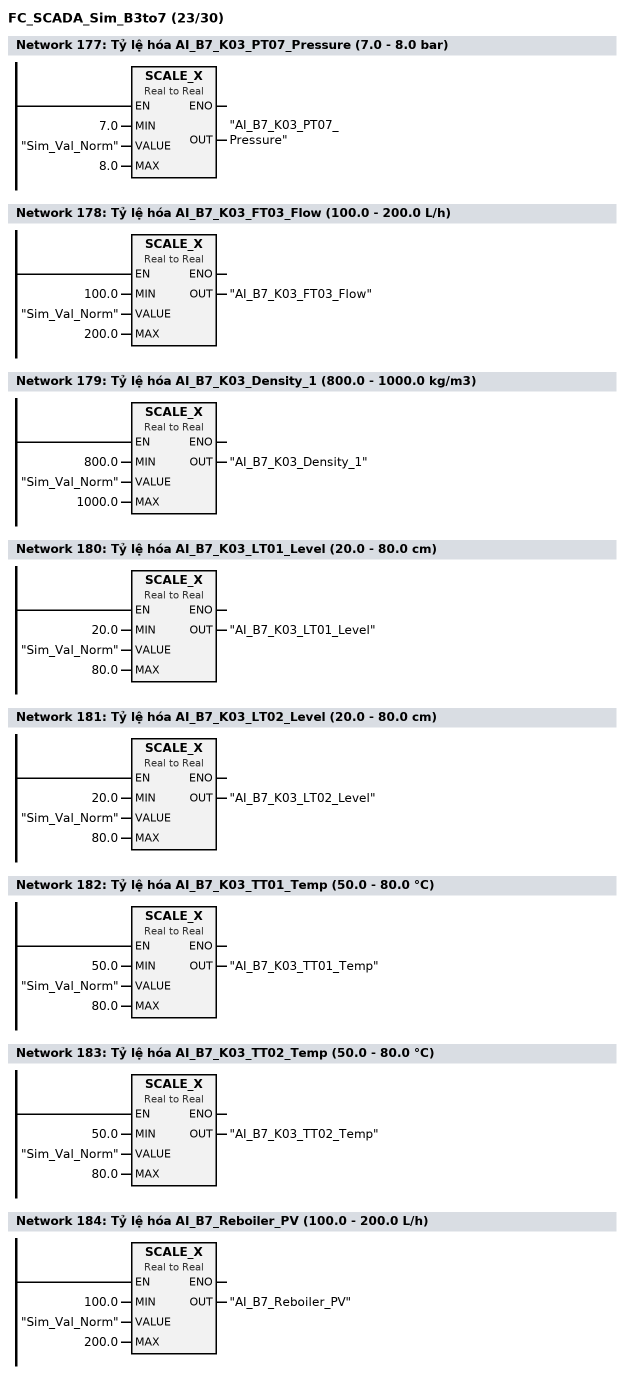
   RUNG wire#powerrail
      { S7_Templates := "[SrcType := Real, DestType := Real]" } Scale(min := 7.0, value := "Sim_Val_Norm", max := 8.0, out => "AI_B7_K03_PT07_Pressure")
   END_RUNG
   // the same network as SCL:
   "AI_B7_K03_PT07_Pressure" := SCALE_X(MIN := 7.0, VALUE := "Sim_Val_Norm", MAX := 8.0);
END_REGION

REGION Network 178: Tỷ lệ hóa AI_B7_K03_FT03_Flow (100.0 - 200.0 L/h)
   RUNG wire#powerrail
      { S7_Templates := "[SrcType := Real, DestType := Real]" } Scale(min := 100.0, value := "Sim_Val_Norm", max := 200.0, out => "AI_B7_K03_FT03_Flow")
   END_RUNG
   // the same network as SCL:
   "AI_B7_K03_FT03_Flow" := SCALE_X(MIN := 100.0, VALUE := "Sim_Val_Norm", MAX := 200.0);
END_REGION

REGION Network 179: Tỷ lệ hóa AI_B7_K03_Density_1 (800.0 - 1000.0 kg/m3)
   RUNG wire#powerrail
      { S7_Templates := "[SrcType := Real, DestType := Real]" } Scale(min := 800.0, value := "Sim_Val_Norm", max := 1000.0, out => "AI_B7_K03_Density_1")
   END_RUNG
   // the same network as SCL:
   "AI_B7_K03_Density_1" := SCALE_X(MIN := 800.0, VALUE := "Sim_Val_Norm", MAX := 1000.0);
END_REGION

REGION Network 180: Tỷ lệ hóa AI_B7_K03_LT01_Level (20.0 - 80.0 cm)
   RUNG wire#powerrail
      { S7_Templates := "[SrcType := Real, DestType := Real]" } Scale(min := 20.0, value := "Sim_Val_Norm", max := 80.0, out => "AI_B7_K03_LT01_Level")
   END_RUNG
   // the same network as SCL:
   "AI_B7_K03_LT01_Level" := SCALE_X(MIN := 20.0, VALUE := "Sim_Val_Norm", MAX := 80.0);
END_REGION

REGION Network 181: Tỷ lệ hóa AI_B7_K03_LT02_Level (20.0 - 80.0 cm)
   RUNG wire#powerrail
      { S7_Templates := "[SrcType := Real, DestType := Real]" } Scale(min := 20.0, value := "Sim_Val_Norm", max := 80.0, out => "AI_B7_K03_LT02_Level")
   END_RUNG
   // the same network as SCL:
   "AI_B7_K03_LT02_Level" := SCALE_X(MIN := 20.0, VALUE := "Sim_Val_Norm", MAX := 80.0);
END_REGION

REGION Network 182: Tỷ lệ hóa AI_B7_K03_TT01_Temp (50.0 - 80.0 °C)
   RUNG wire#powerrail
      { S7_Templates := "[SrcType := Real, DestType := Real]" } Scale(min := 50.0, value := "Sim_Val_Norm", max := 80.0, out => "AI_B7_K03_TT01_Temp")
   END_RUNG
   // the same network as SCL:
   "AI_B7_K03_TT01_Temp" := SCALE_X(MIN := 50.0, VALUE := "Sim_Val_Norm", MAX := 80.0);
END_REGION

REGION Network 183: Tỷ lệ hóa AI_B7_K03_TT02_Temp (50.0 - 80.0 °C)
   RUNG wire#powerrail
      { S7_Templates := "[SrcType := Real, DestType := Real]" } Scale(min := 50.0, value := "Sim_Val_Norm", max := 80.0, out => "AI_B7_K03_TT02_Temp")
   END_RUNG
   // the same network as SCL:
   "AI_B7_K03_TT02_Temp" := SCALE_X(MIN := 50.0, VALUE := "Sim_Val_Norm", MAX := 80.0);
END_REGION

REGION Network 184: Tỷ lệ hóa AI_B7_Reboiler_PV (100.0 - 200.0 L/h)
   RUNG wire#powerrail
      { S7_Templates := "[SrcType := Real, DestType := Real]" } Scale(min := 100.0, value := "Sim_Val_Norm", max := 200.0, out => "AI_B7_Reboiler_PV")
   END_RUNG
   // the same network as SCL:
   "AI_B7_Reboiler_PV" := SCALE_X(MIN := 100.0, VALUE := "Sim_Val_Norm", MAX := 200.0);
END_REGION

REGION Network 185: Tỷ lệ hóa AI_B7_Reboiler_SP (100.0 - 200.0 L/h)
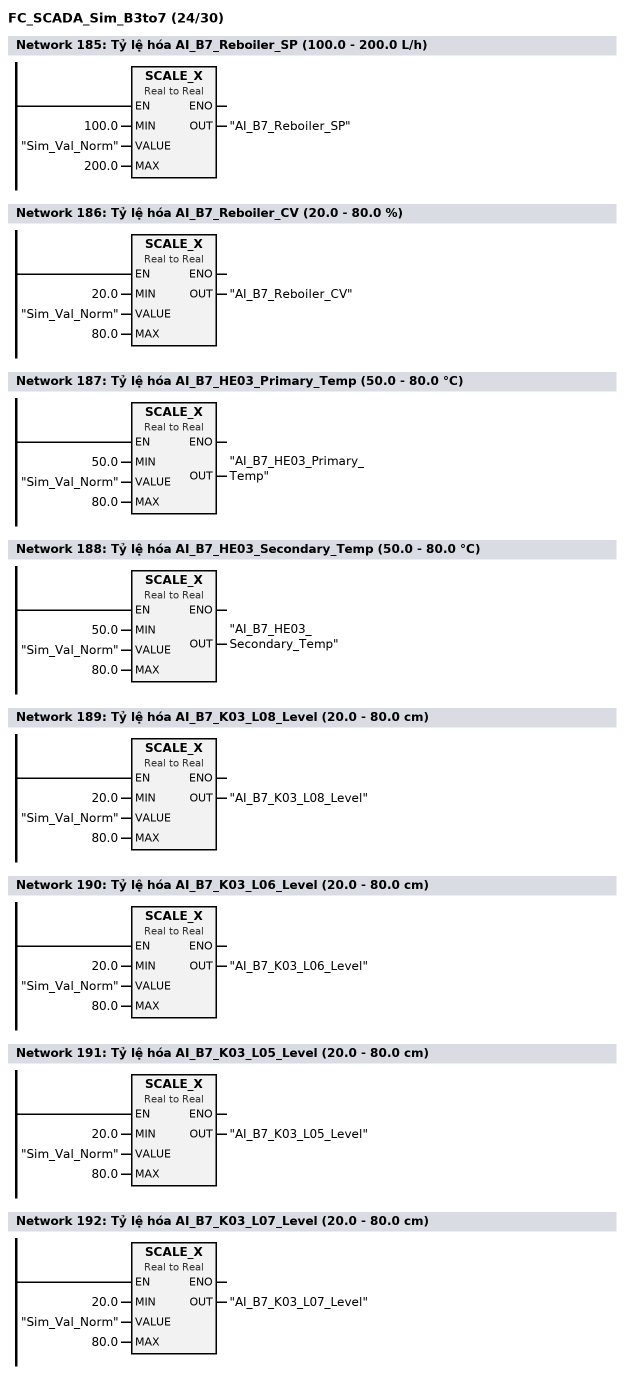
   RUNG wire#powerrail
      { S7_Templates := "[SrcType := Real, DestType := Real]" } Scale(min := 100.0, value := "Sim_Val_Norm", max := 200.0, out => "AI_B7_Reboiler_SP")
   END_RUNG
   // the same network as SCL:
   "AI_B7_Reboiler_SP" := SCALE_X(MIN := 100.0, VALUE := "Sim_Val_Norm", MAX := 200.0);
END_REGION

REGION Network 186: Tỷ lệ hóa AI_B7_Reboiler_CV (20.0 - 80.0 %)
   RUNG wire#powerrail
      { S7_Templates := "[SrcType := Real, DestType := Real]" } Scale(min := 20.0, value := "Sim_Val_Norm", max := 80.0, out => "AI_B7_Reboiler_CV")
   END_RUNG
   // the same network as SCL:
   "AI_B7_Reboiler_CV" := SCALE_X(MIN := 20.0, VALUE := "Sim_Val_Norm", MAX := 80.0);
END_REGION

REGION Network 187: Tỷ lệ hóa AI_B7_HE03_Primary_Temp (50.0 - 80.0 °C)
   RUNG wire#powerrail
      { S7_Templates := "[SrcType := Real, DestType := Real]" } Scale(min := 50.0, value := "Sim_Val_Norm", max := 80.0, out => "AI_B7_HE03_Primary_Temp")
   END_RUNG
   // the same network as SCL:
   "AI_B7_HE03_Primary_Temp" := SCALE_X(MIN := 50.0, VALUE := "Sim_Val_Norm", MAX := 80.0);
END_REGION

REGION Network 188: Tỷ lệ hóa AI_B7_HE03_Secondary_Temp (50.0 - 80.0 °C)
   RUNG wire#powerrail
      { S7_Templates := "[SrcType := Real, DestType := Real]" } Scale(min := 50.0, value := "Sim_Val_Norm", max := 80.0, out => "AI_B7_HE03_Secondary_Temp")
   END_RUNG
   // the same network as SCL:
   "AI_B7_HE03_Secondary_Temp" := SCALE_X(MIN := 50.0, VALUE := "Sim_Val_Norm", MAX := 80.0);
END_REGION

REGION Network 189: Tỷ lệ hóa AI_B7_K03_L08_Level (20.0 - 80.0 cm)
   RUNG wire#powerrail
      { S7_Templates := "[SrcType := Real, DestType := Real]" } Scale(min := 20.0, value := "Sim_Val_Norm", max := 80.0, out => "AI_B7_K03_L08_Level")
   END_RUNG
   // the same network as SCL:
   "AI_B7_K03_L08_Level" := SCALE_X(MIN := 20.0, VALUE := "Sim_Val_Norm", MAX := 80.0);
END_REGION

REGION Network 190: Tỷ lệ hóa AI_B7_K03_L06_Level (20.0 - 80.0 cm)
   RUNG wire#powerrail
      { S7_Templates := "[SrcType := Real, DestType := Real]" } Scale(min := 20.0, value := "Sim_Val_Norm", max := 80.0, out => "AI_B7_K03_L06_Level")
   END_RUNG
   // the same network as SCL:
   "AI_B7_K03_L06_Level" := SCALE_X(MIN := 20.0, VALUE := "Sim_Val_Norm", MAX := 80.0);
END_REGION

REGION Network 191: Tỷ lệ hóa AI_B7_K03_L05_Level (20.0 - 80.0 cm)
   RUNG wire#powerrail
      { S7_Templates := "[SrcType := Real, DestType := Real]" } Scale(min := 20.0, value := "Sim_Val_Norm", max := 80.0, out => "AI_B7_K03_L05_Level")
   END_RUNG
   // the same network as SCL:
   "AI_B7_K03_L05_Level" := SCALE_X(MIN := 20.0, VALUE := "Sim_Val_Norm", MAX := 80.0);
END_REGION

REGION Network 192: Tỷ lệ hóa AI_B7_K03_L07_Level (20.0 - 80.0 cm)
   RUNG wire#powerrail
      { S7_Templates := "[SrcType := Real, DestType := Real]" } Scale(min := 20.0, value := "Sim_Val_Norm", max := 80.0, out => "AI_B7_K03_L07_Level")
   END_RUNG
   // the same network as SCL:
   "AI_B7_K03_L07_Level" := SCALE_X(MIN := 20.0, VALUE := "Sim_Val_Norm", MAX := 80.0);
END_REGION

REGION Network 193: Tỷ lệ hóa AI_B7_K03_L04_Level (20.0 - 80.0 cm)
